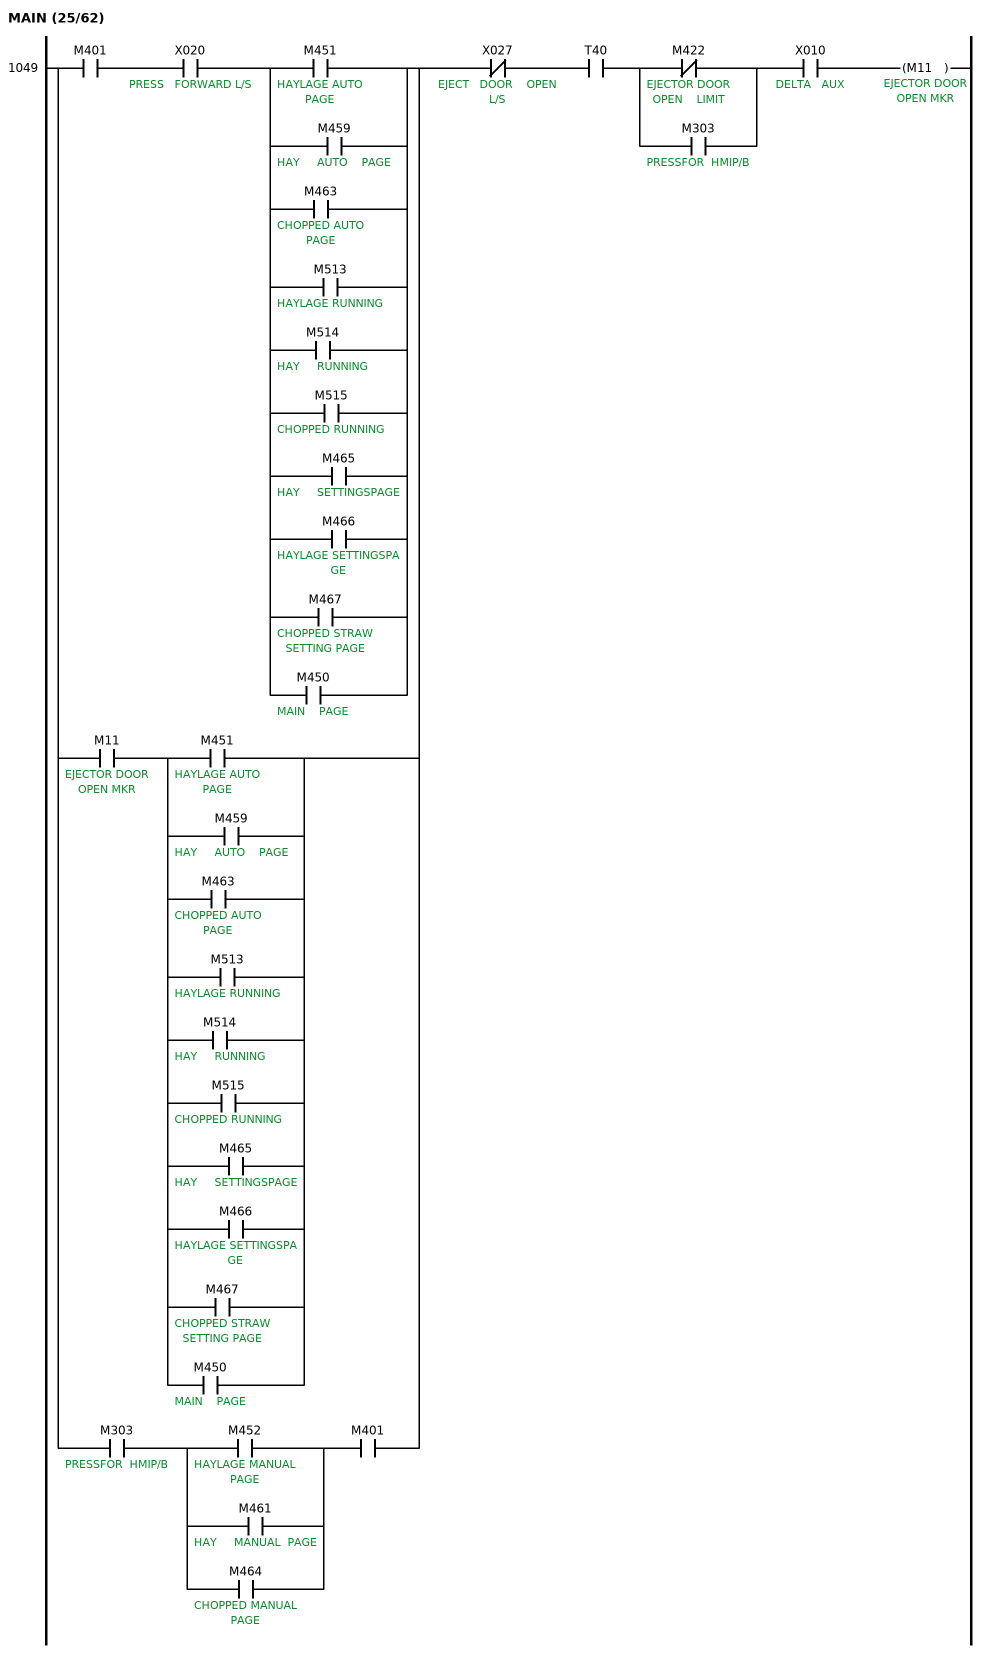
1049  LD      M401
      AND     X020  ; PRESS   FORWARD L/S
      LD      M451  ; HAYLAGE AUTO    PAGE
      OR      M459  ; HAY     AUTO    PAGE
      OR      M463  ; CHOPPED AUTO    PAGE
      OR      M513  ; HAYLAGE RUNNING
      OR      M514  ; HAY     RUNNING
      OR      M515  ; CHOPPED RUNNING
      OR      M465  ; HAY     SETTINGSPAGE
      OR      M466  ; HAYLAGE SETTINGSPAGE
      OR      M467  ; CHOPPED STRAW   SETTING PAGE
      OR      M450  ; MAIN    PAGE
      ANB
      LD      M11  ; EJECTOR DOOR    OPEN MKR
      LD      M451  ; HAYLAGE AUTO    PAGE
      OR      M459  ; HAY     AUTO    PAGE
      OR      M463  ; CHOPPED AUTO    PAGE
      OR      M513  ; HAYLAGE RUNNING
      OR      M514  ; HAY     RUNNING
      OR      M515  ; CHOPPED RUNNING
      OR      M465  ; HAY     SETTINGSPAGE
      OR      M466  ; HAYLAGE SETTINGSPAGE
      OR      M467  ; CHOPPED STRAW   SETTING PAGE
      OR      M450  ; MAIN    PAGE
      ANB
      ORB
      LD      M303  ; PRESSFOR  HMIP/B
      LD      M452  ; HAYLAGE MANUAL  PAGE
      OR      M461  ; HAY     MANUAL  PAGE
      OR      M464  ; CHOPPED MANUAL  PAGE
      ANB
      AND     M401
      ORB
      ANI     X027  ; EJECT   DOOR    OPEN L/S
      AND     T40
      LDI     M422  ; EJECTOR DOOR    OPEN    LIMIT
      OR      M303  ; PRESSFOR  HMIP/B
      ANB
      AND     X010  ; DELTA   AUX
      OUT     M11  ; EJECTOR DOOR    OPEN MKR
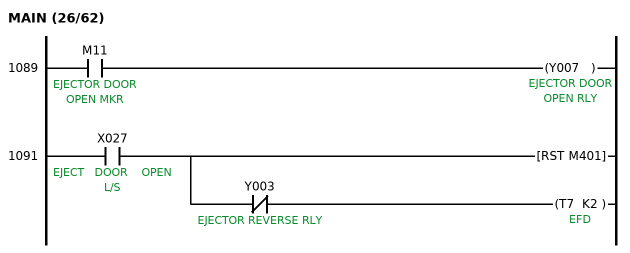
1089  LD      M11  ; EJECTOR DOOR    OPEN MKR
      OUT     Y007  ; EJECTOR DOOR    OPEN RLY
1091  LD      X027  ; EJECT   DOOR    OPEN L/S
      RST     M401
      ANI     Y003  ; EJECTOR REVERSE RLY
      OUT     T7 K2  ; EFD
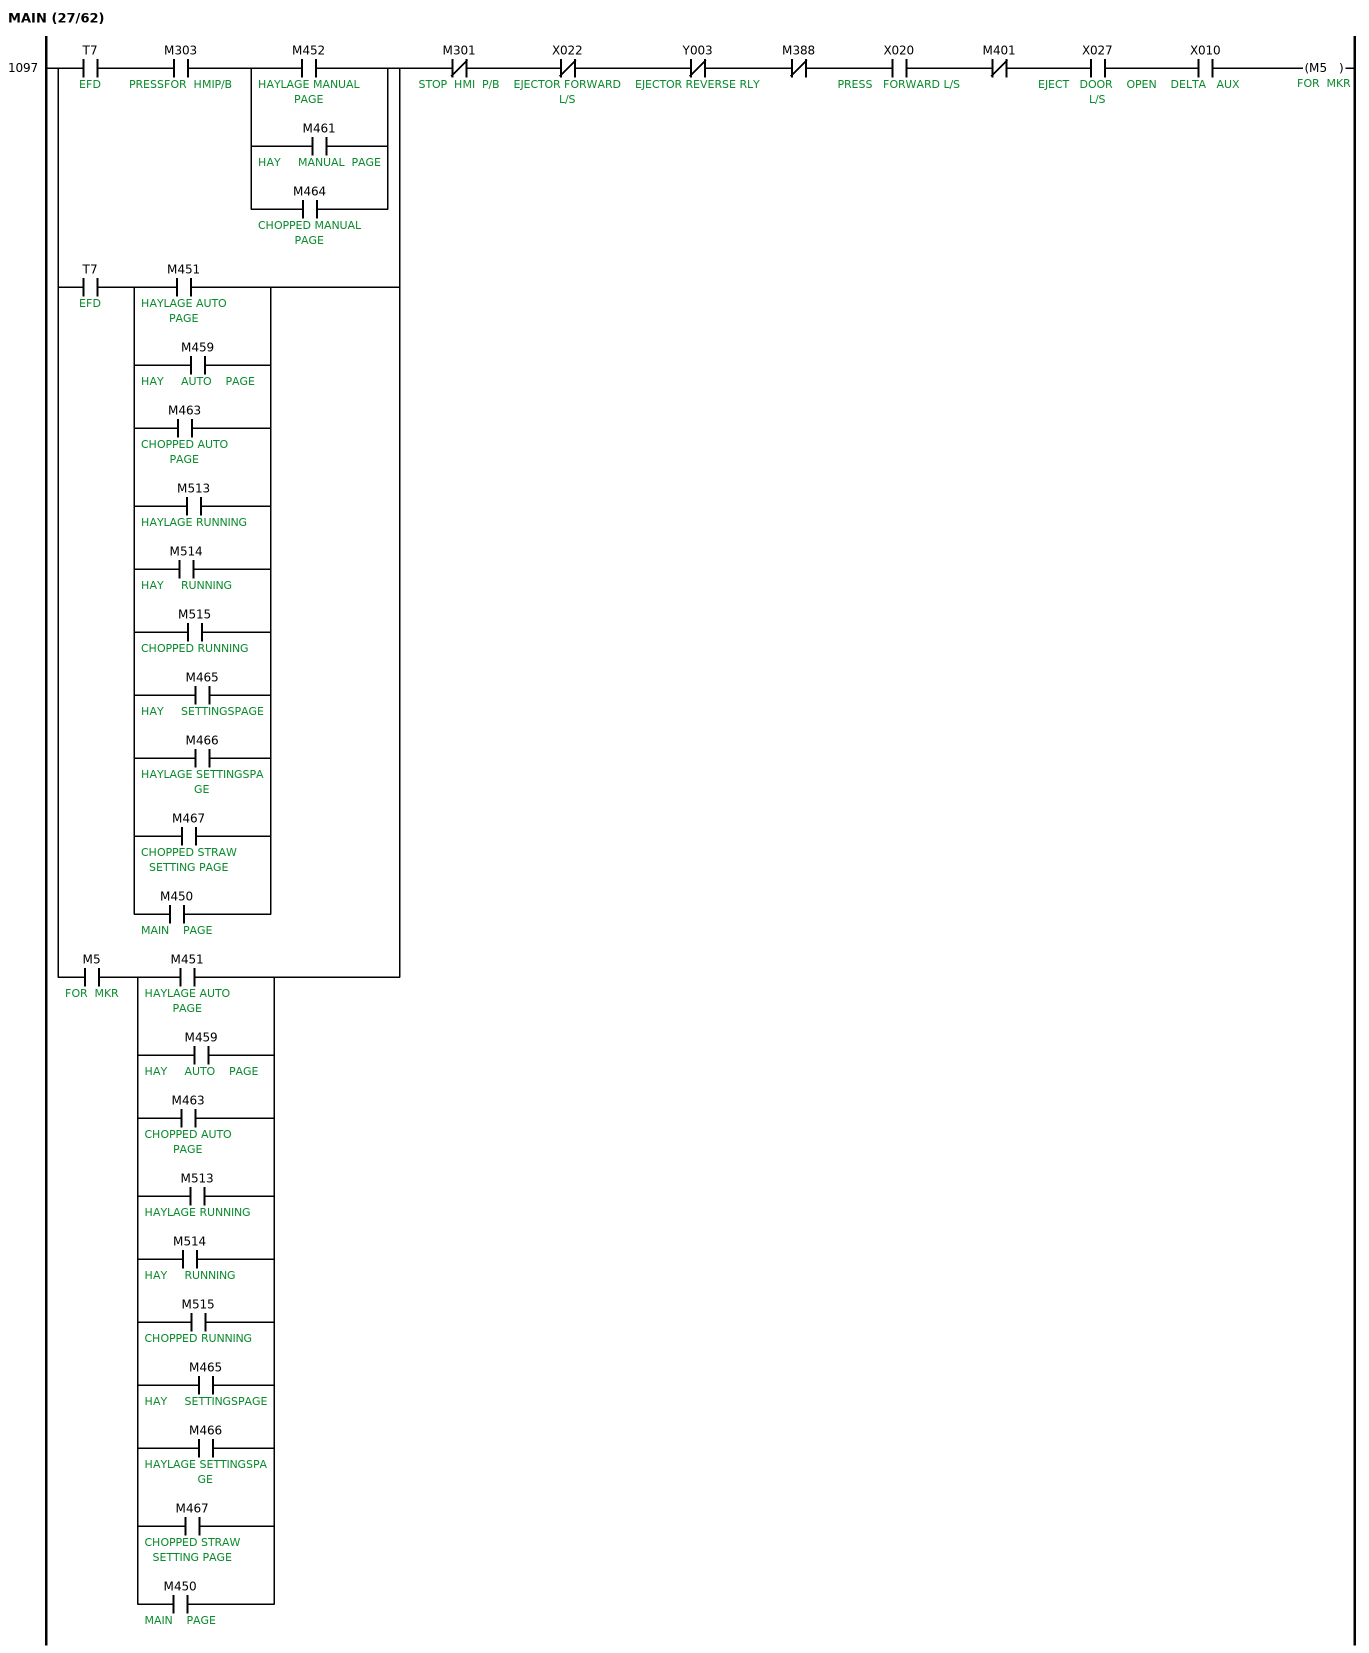
1097  LD      T7  ; EFD
      AND     M303  ; PRESSFOR  HMIP/B
      LD      M452  ; HAYLAGE MANUAL  PAGE
      OR      M461  ; HAY     MANUAL  PAGE
      OR      M464  ; CHOPPED MANUAL  PAGE
      ANB
      LD      T7  ; EFD
      LD      M451  ; HAYLAGE AUTO    PAGE
      OR      M459  ; HAY     AUTO    PAGE
      OR      M463  ; CHOPPED AUTO    PAGE
      OR      M513  ; HAYLAGE RUNNING
      OR      M514  ; HAY     RUNNING
      OR      M515  ; CHOPPED RUNNING
      OR      M465  ; HAY     SETTINGSPAGE
      OR      M466  ; HAYLAGE SETTINGSPAGE
      OR      M467  ; CHOPPED STRAW   SETTING PAGE
      OR      M450  ; MAIN    PAGE
      ANB
      ORB
      LD      M5  ; FOR  MKR
      LD      M451  ; HAYLAGE AUTO    PAGE
      OR      M459  ; HAY     AUTO    PAGE
      OR      M463  ; CHOPPED AUTO    PAGE
      OR      M513  ; HAYLAGE RUNNING
      OR      M514  ; HAY     RUNNING
      OR      M515  ; CHOPPED RUNNING
      OR      M465  ; HAY     SETTINGSPAGE
      OR      M466  ; HAYLAGE SETTINGSPAGE
      OR      M467  ; CHOPPED STRAW   SETTING PAGE
      OR      M450  ; MAIN    PAGE
      ANB
      ORB
      ANI     M301  ; STOP  HMI  P/B
      ANI     X022  ; EJECTOR FORWARD L/S
      ANI     Y003  ; EJECTOR REVERSE RLY
      ANI     M388
      AND     X020  ; PRESS   FORWARD L/S
      ANI     M401
      AND     X027  ; EJECT   DOOR    OPEN L/S
      AND     X010  ; DELTA   AUX
      OUT     M5  ; FOR  MKR
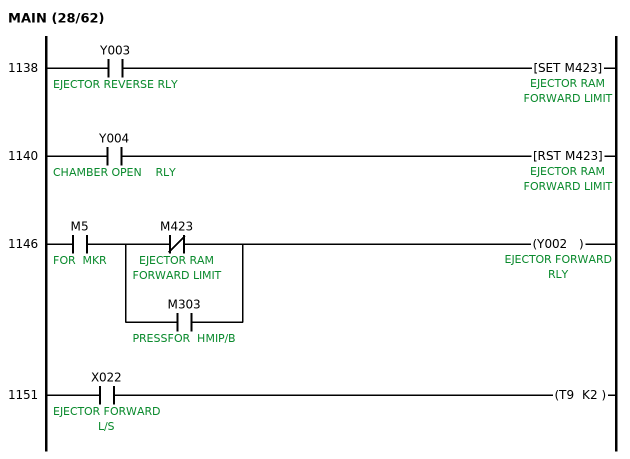
1138  LD      Y003  ; EJECTOR REVERSE RLY
      SET     M423  ; EJECTOR RAM     FORWARD LIMIT
1140  LD      Y004  ; CHAMBER OPEN    RLY
      RST     M423  ; EJECTOR RAM     FORWARD LIMIT
1146  LD      M5  ; FOR  MKR
      LDI     M423  ; EJECTOR RAM     FORWARD LIMIT
      OR      M303  ; PRESSFOR  HMIP/B
      ANB
      OUT     Y002  ; EJECTOR FORWARD RLY
1151  LD      X022  ; EJECTOR FORWARD L/S
      OUT     T9 K2
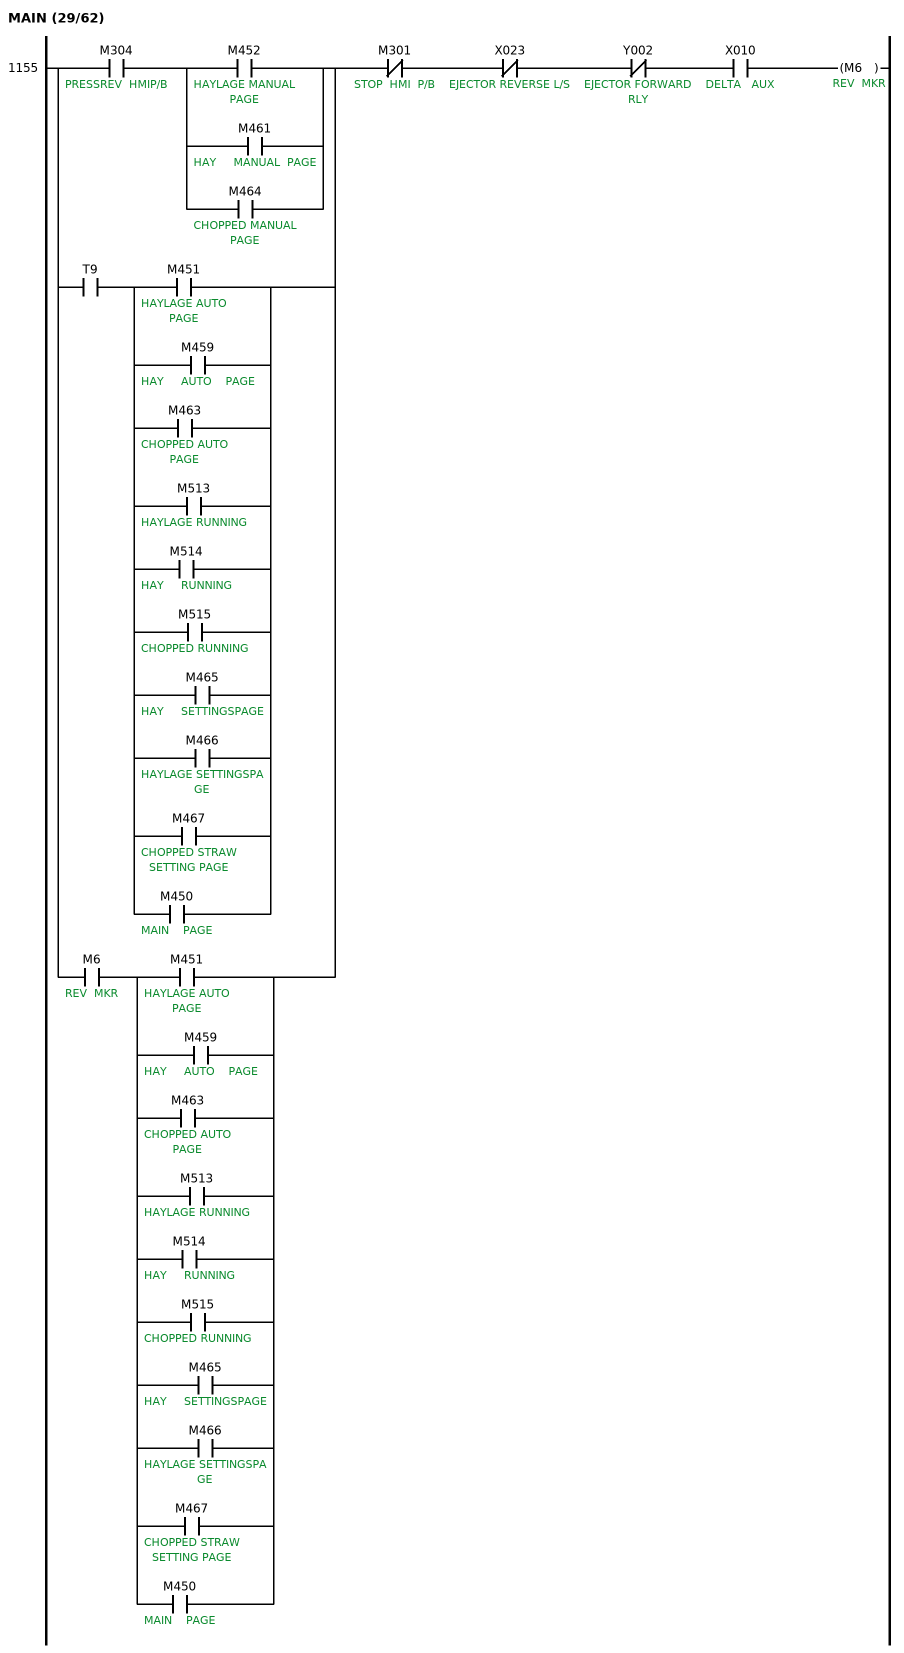
1155  LD      M304  ; PRESSREV  HMIP/B
      LD      M452  ; HAYLAGE MANUAL  PAGE
      OR      M461  ; HAY     MANUAL  PAGE
      OR      M464  ; CHOPPED MANUAL  PAGE
      ANB
      LD      T9
      LD      M451  ; HAYLAGE AUTO    PAGE
      OR      M459  ; HAY     AUTO    PAGE
      OR      M463  ; CHOPPED AUTO    PAGE
      OR      M513  ; HAYLAGE RUNNING
      OR      M514  ; HAY     RUNNING
      OR      M515  ; CHOPPED RUNNING
      OR      M465  ; HAY     SETTINGSPAGE
      OR      M466  ; HAYLAGE SETTINGSPAGE
      OR      M467  ; CHOPPED STRAW   SETTING PAGE
      OR      M450  ; MAIN    PAGE
      ANB
      ORB
      LD      M6  ; REV  MKR
      LD      M451  ; HAYLAGE AUTO    PAGE
      OR      M459  ; HAY     AUTO    PAGE
      OR      M463  ; CHOPPED AUTO    PAGE
      OR      M513  ; HAYLAGE RUNNING
      OR      M514  ; HAY     RUNNING
      OR      M515  ; CHOPPED RUNNING
      OR      M465  ; HAY     SETTINGSPAGE
      OR      M466  ; HAYLAGE SETTINGSPAGE
      OR      M467  ; CHOPPED STRAW   SETTING PAGE
      OR      M450  ; MAIN    PAGE
      ANB
      ORB
      ANI     M301  ; STOP  HMI  P/B
      ANI     X023  ; EJECTOR REVERSE L/S
      ANI     Y002  ; EJECTOR FORWARD RLY
      AND     X010  ; DELTA   AUX
      OUT     M6  ; REV  MKR
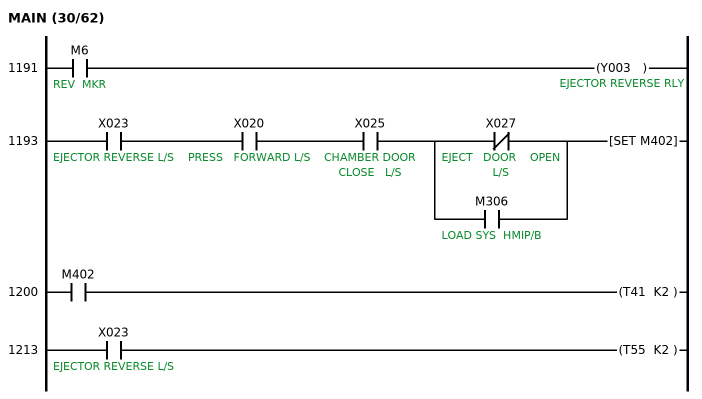
1191  LD      M6  ; REV  MKR
      OUT     Y003  ; EJECTOR REVERSE RLY
1193  LD      X023  ; EJECTOR REVERSE L/S
      AND     X020  ; PRESS   FORWARD L/S
      AND     X025  ; CHAMBER DOOR    CLOSE   L/S
      LDI     X027  ; EJECT   DOOR    OPEN L/S
      OR      M306  ; LOAD SYS  HMIP/B
      ANB
      SET     M402
1200  LD      M402
      OUT     T41 K2
1213  LD      X023  ; EJECTOR REVERSE L/S
      OUT     T55 K2
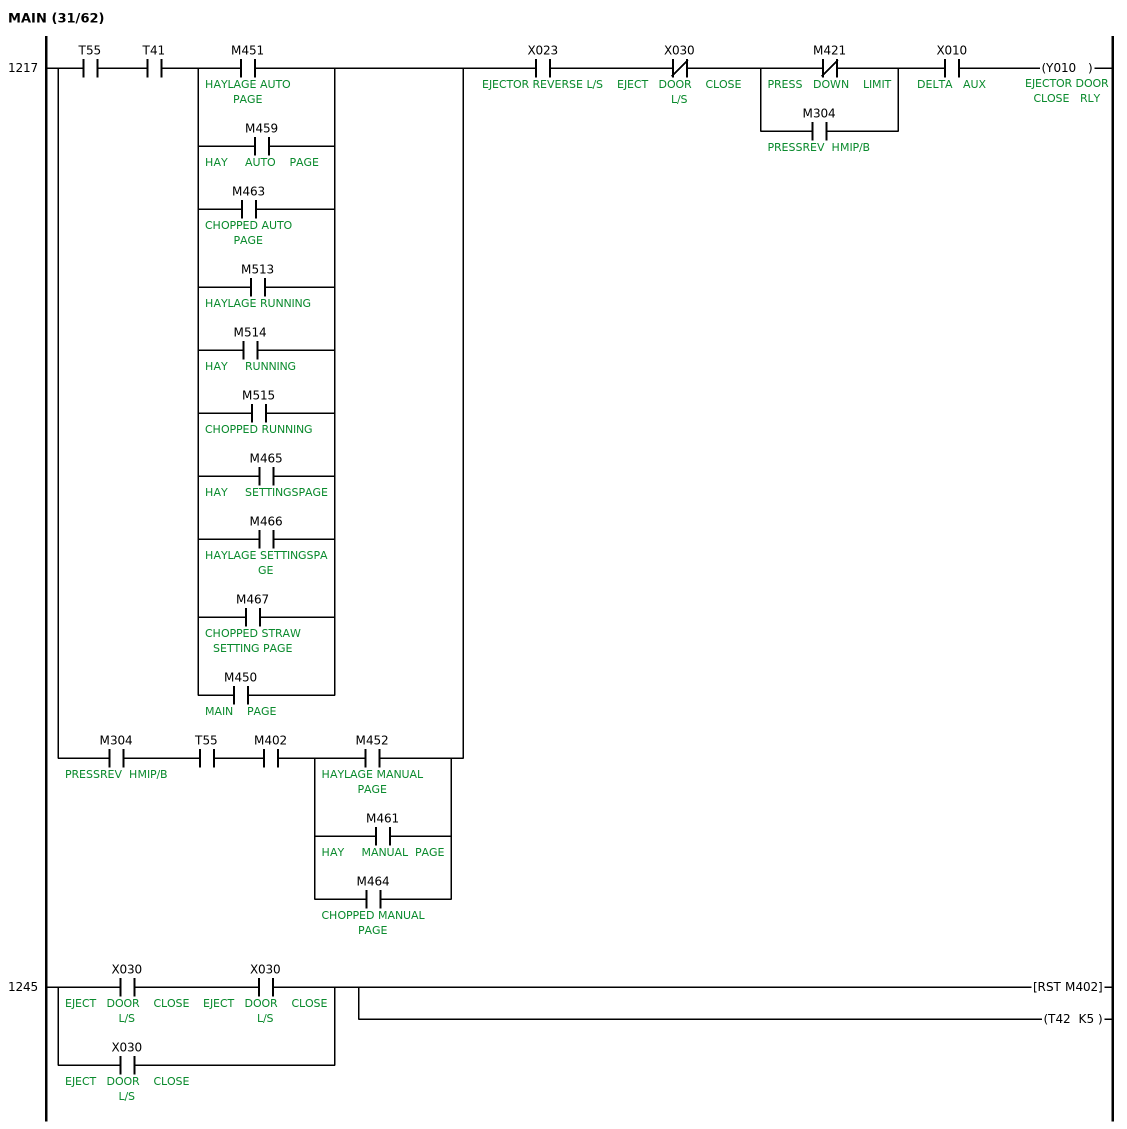
1217  LD      T55
      AND     T41
      LD      M451  ; HAYLAGE AUTO    PAGE
      OR      M459  ; HAY     AUTO    PAGE
      OR      M463  ; CHOPPED AUTO    PAGE
      OR      M513  ; HAYLAGE RUNNING
      OR      M514  ; HAY     RUNNING
      OR      M515  ; CHOPPED RUNNING
      OR      M465  ; HAY     SETTINGSPAGE
      OR      M466  ; HAYLAGE SETTINGSPAGE
      OR      M467  ; CHOPPED STRAW   SETTING PAGE
      OR      M450  ; MAIN    PAGE
      ANB
      LD      M304  ; PRESSREV  HMIP/B
      AND     T55
      AND     M402
      LD      M452  ; HAYLAGE MANUAL  PAGE
      OR      M461  ; HAY     MANUAL  PAGE
      OR      M464  ; CHOPPED MANUAL  PAGE
      ANB
      ORB
      AND     X023  ; EJECTOR REVERSE L/S
      ANI     X030  ; EJECT   DOOR    CLOSE L/S
      LDI     M421  ; PRESS   DOWN    LIMIT
      OR      M304  ; PRESSREV  HMIP/B
      ANB
      AND     X010  ; DELTA   AUX
      OUT     Y010  ; EJECTOR DOOR    CLOSE   RLY
1245  LD      X030  ; EJECT   DOOR    CLOSE L/S
      AND     X030  ; EJECT   DOOR    CLOSE L/S
      OR      X030  ; EJECT   DOOR    CLOSE L/S
      RST     M402
      OUT     T42 K5
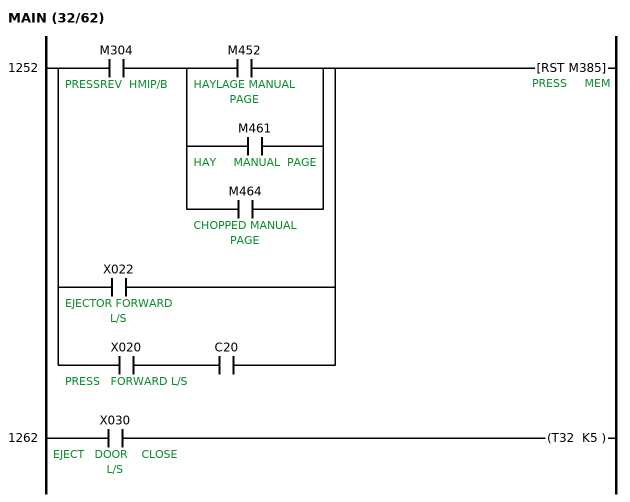
1252  LD      M304  ; PRESSREV  HMIP/B
      LD      M452  ; HAYLAGE MANUAL  PAGE
      OR      M461  ; HAY     MANUAL  PAGE
      OR      M464  ; CHOPPED MANUAL  PAGE
      ANB
      OR      X022  ; EJECTOR FORWARD L/S
      LD      X020  ; PRESS   FORWARD L/S
      AND     C20
      ORB
      RST     M385  ; PRESS     MEM
1262  LD      X030  ; EJECT   DOOR    CLOSE L/S
      OUT     T32 K5
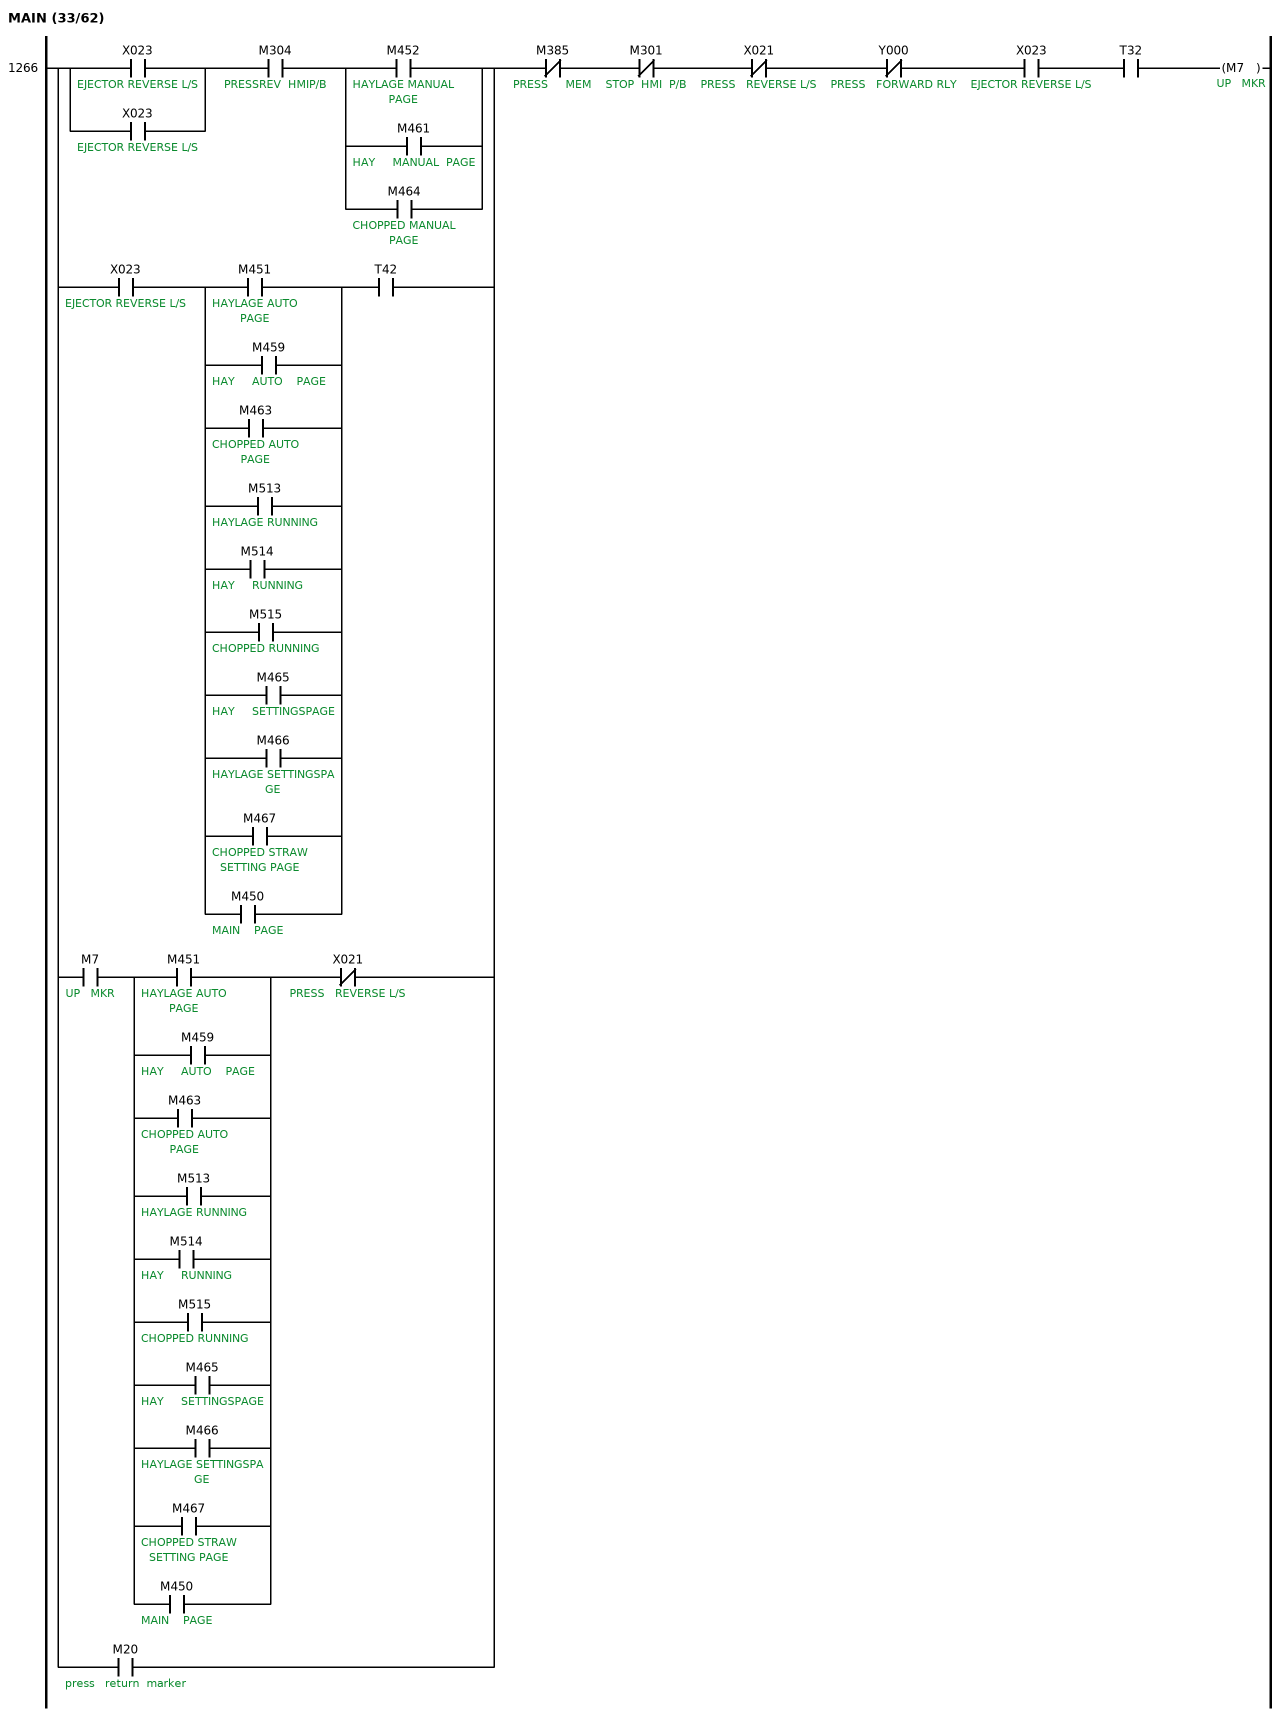
1266  LD      X023  ; EJECTOR REVERSE L/S
      OR      X023  ; EJECTOR REVERSE L/S
      AND     M304  ; PRESSREV  HMIP/B
      LD      M452  ; HAYLAGE MANUAL  PAGE
      OR      M461  ; HAY     MANUAL  PAGE
      OR      M464  ; CHOPPED MANUAL  PAGE
      ANB
      LD      X023  ; EJECTOR REVERSE L/S
      LD      M451  ; HAYLAGE AUTO    PAGE
      OR      M459  ; HAY     AUTO    PAGE
      OR      M463  ; CHOPPED AUTO    PAGE
      OR      M513  ; HAYLAGE RUNNING
      OR      M514  ; HAY     RUNNING
      OR      M515  ; CHOPPED RUNNING
      OR      M465  ; HAY     SETTINGSPAGE
      OR      M466  ; HAYLAGE SETTINGSPAGE
      OR      M467  ; CHOPPED STRAW   SETTING PAGE
      OR      M450  ; MAIN    PAGE
      ANB
      AND     T42
      ORB
      LD      M7  ; UP   MKR
      LD      M451  ; HAYLAGE AUTO    PAGE
      OR      M459  ; HAY     AUTO    PAGE
      OR      M463  ; CHOPPED AUTO    PAGE
      OR      M513  ; HAYLAGE RUNNING
      OR      M514  ; HAY     RUNNING
      OR      M515  ; CHOPPED RUNNING
      OR      M465  ; HAY     SETTINGSPAGE
      OR      M466  ; HAYLAGE SETTINGSPAGE
      OR      M467  ; CHOPPED STRAW   SETTING PAGE
      OR      M450  ; MAIN    PAGE
      ANB
      ANI     X021  ; PRESS   REVERSE L/S
      ORB
      OR      M20  ; press   return  marker
      ANI     M385  ; PRESS     MEM
      ANI     M301  ; STOP  HMI  P/B
      ANI     X021  ; PRESS   REVERSE L/S
      ANI     Y000  ; PRESS   FORWARD RLY
      AND     X023  ; EJECTOR REVERSE L/S
      AND     T32
      OUT     M7  ; UP   MKR
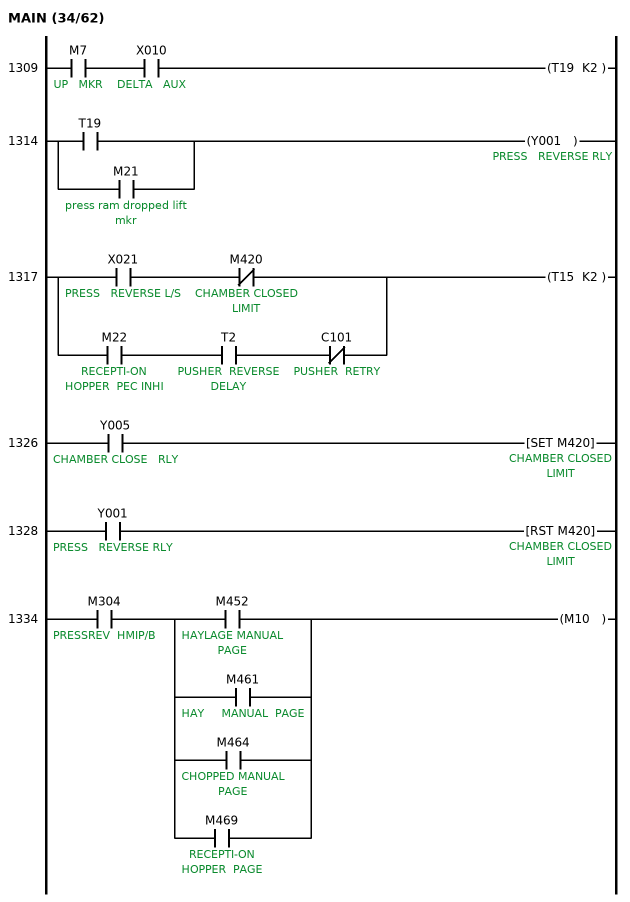
1309  LD      M7  ; UP   MKR
      AND     X010  ; DELTA   AUX
      OUT     T19 K2
1314  LD      T19
      OR      M21  ; press ram dropped lift mkr
      OUT     Y001  ; PRESS   REVERSE RLY
1317  LD      X021  ; PRESS   REVERSE L/S
      ANI     M420  ; CHAMBER CLOSED  LIMIT
      LD      M22  ; RECEPTI-ON      HOPPER  PEC INHI
      AND     T2  ; PUSHER  REVERSE DELAY
      ANI     C101  ; PUSHER  RETRY
      ORB
      OUT     T15 K2
1326  LD      Y005  ; CHAMBER CLOSE   RLY
      SET     M420  ; CHAMBER CLOSED  LIMIT
1328  LD      Y001  ; PRESS   REVERSE RLY
      RST     M420  ; CHAMBER CLOSED  LIMIT
1334  LD      M304  ; PRESSREV  HMIP/B
      LD      M452  ; HAYLAGE MANUAL  PAGE
      OR      M461  ; HAY     MANUAL  PAGE
      OR      M464  ; CHOPPED MANUAL  PAGE
      OR      M469  ; RECEPTI-ON      HOPPER  PAGE
      ANB
      OUT     M10
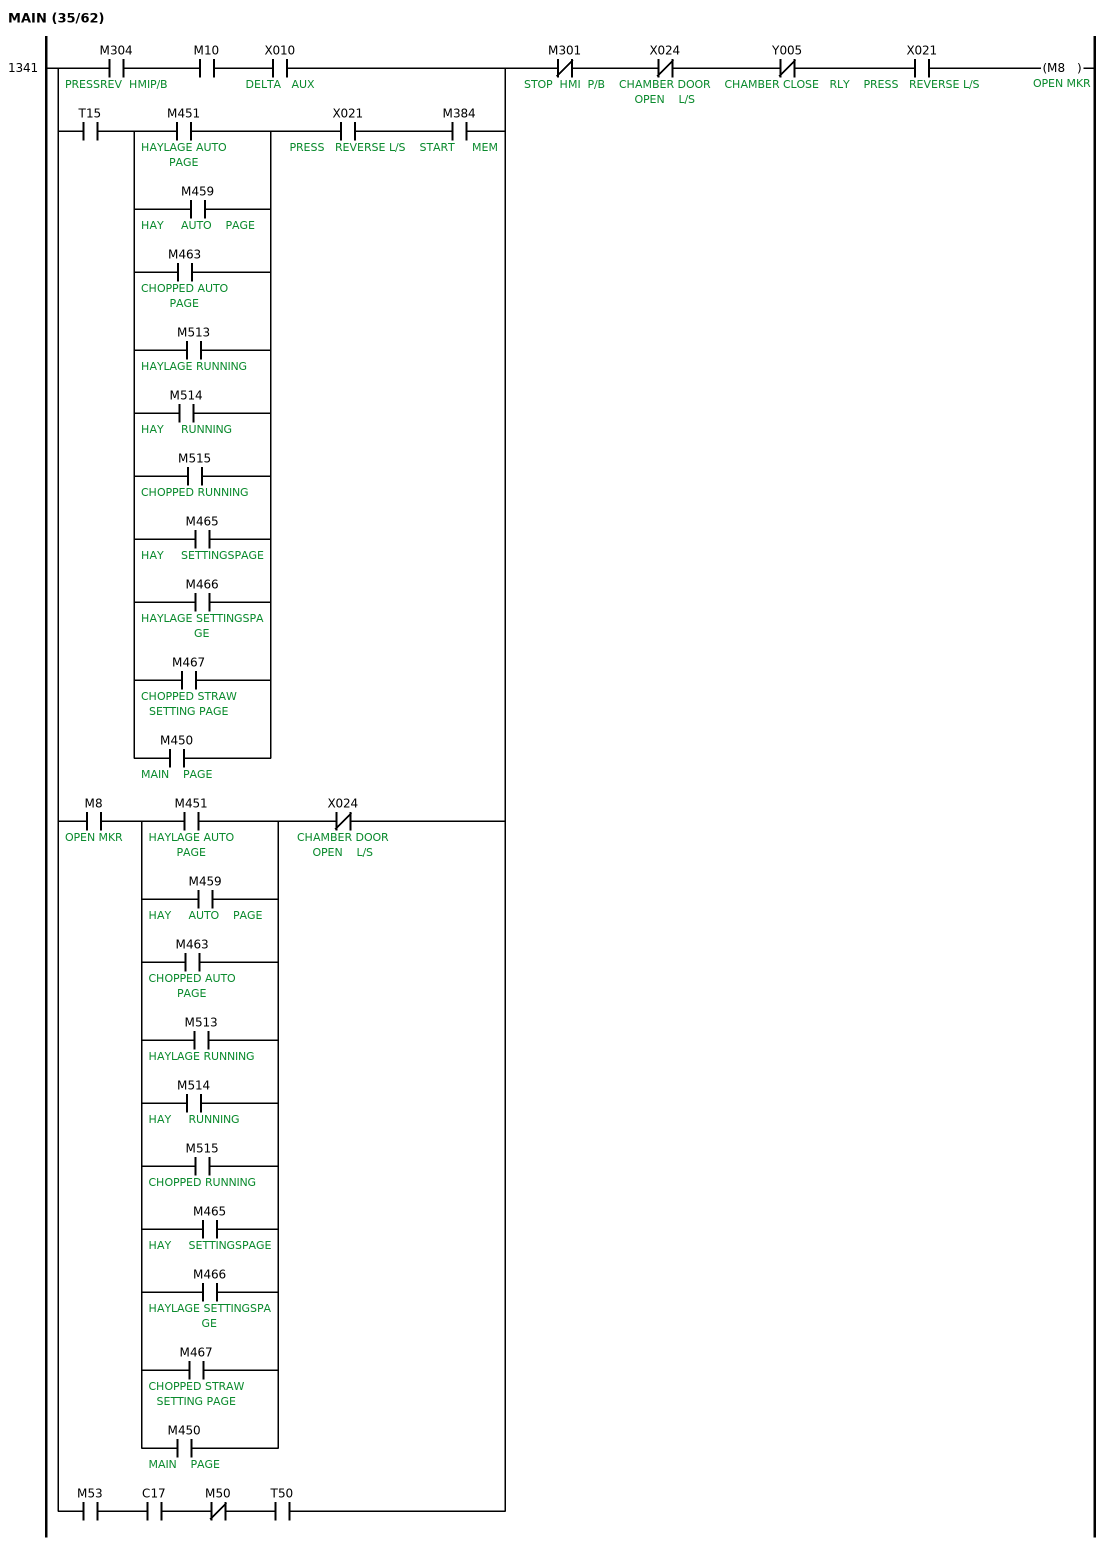
1341  LD      M304  ; PRESSREV  HMIP/B
      AND     M10
      AND     X010  ; DELTA   AUX
      LD      T15
      LD      M451  ; HAYLAGE AUTO    PAGE
      OR      M459  ; HAY     AUTO    PAGE
      OR      M463  ; CHOPPED AUTO    PAGE
      OR      M513  ; HAYLAGE RUNNING
      OR      M514  ; HAY     RUNNING
      OR      M515  ; CHOPPED RUNNING
      OR      M465  ; HAY     SETTINGSPAGE
      OR      M466  ; HAYLAGE SETTINGSPAGE
      OR      M467  ; CHOPPED STRAW   SETTING PAGE
      OR      M450  ; MAIN    PAGE
      ANB
      AND     X021  ; PRESS   REVERSE L/S
      AND     M384  ; START     MEM
      ORB
      LD      M8  ; OPEN MKR
      LD      M451  ; HAYLAGE AUTO    PAGE
      OR      M459  ; HAY     AUTO    PAGE
      OR      M463  ; CHOPPED AUTO    PAGE
      OR      M513  ; HAYLAGE RUNNING
      OR      M514  ; HAY     RUNNING
      OR      M515  ; CHOPPED RUNNING
      OR      M465  ; HAY     SETTINGSPAGE
      OR      M466  ; HAYLAGE SETTINGSPAGE
      OR      M467  ; CHOPPED STRAW   SETTING PAGE
      OR      M450  ; MAIN    PAGE
      ANB
      ANI     X024  ; CHAMBER DOOR    OPEN    L/S
      ORB
      LD      M53
      AND     C17
      ANI     M50
      AND     T50
      ORB
      ANI     M301  ; STOP  HMI  P/B
      ANI     X024  ; CHAMBER DOOR    OPEN    L/S
      ANI     Y005  ; CHAMBER CLOSE   RLY
      AND     X021  ; PRESS   REVERSE L/S
      OUT     M8  ; OPEN MKR
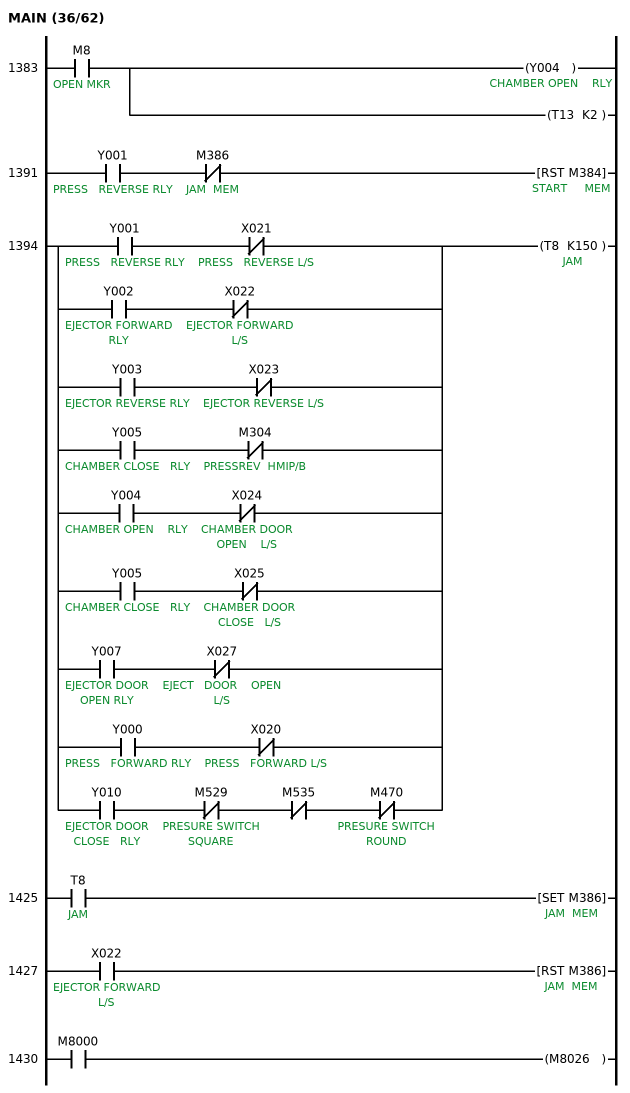
1383  LD      M8  ; OPEN MKR
      OUT     Y004  ; CHAMBER OPEN    RLY
      OUT     T13 K2
1391  LD      Y001  ; PRESS   REVERSE RLY
      ANI     M386  ; JAM  MEM
      RST     M384  ; START     MEM
1394  LD      Y001  ; PRESS   REVERSE RLY
      ANI     X021  ; PRESS   REVERSE L/S
      LD      Y002  ; EJECTOR FORWARD RLY
      ANI     X022  ; EJECTOR FORWARD L/S
      ORB
      LD      Y003  ; EJECTOR REVERSE RLY
      ANI     X023  ; EJECTOR REVERSE L/S
      ORB
      LD      Y005  ; CHAMBER CLOSE   RLY
      ANI     M304  ; PRESSREV  HMIP/B
      ORB
      LD      Y004  ; CHAMBER OPEN    RLY
      ANI     X024  ; CHAMBER DOOR    OPEN    L/S
      ORB
      LD      Y005  ; CHAMBER CLOSE   RLY
      ANI     X025  ; CHAMBER DOOR    CLOSE   L/S
      ORB
      LD      Y007  ; EJECTOR DOOR    OPEN RLY
      ANI     X027  ; EJECT   DOOR    OPEN L/S
      ORB
      LD      Y000  ; PRESS   FORWARD RLY
      ANI     X020  ; PRESS   FORWARD L/S
      ORB
      LD      Y010  ; EJECTOR DOOR    CLOSE   RLY
      ANI     M529  ; PRESURE SWITCH  SQUARE
      ANI     M535
      ANI     M470  ; PRESURE SWITCH  ROUND
      ORB
      OUT     T8 K150  ; JAM
1425  LD      T8  ; JAM
      SET     M386  ; JAM  MEM
1427  LD      X022  ; EJECTOR FORWARD L/S
      RST     M386  ; JAM  MEM
1430  LD      M8000
      OUT     M8026
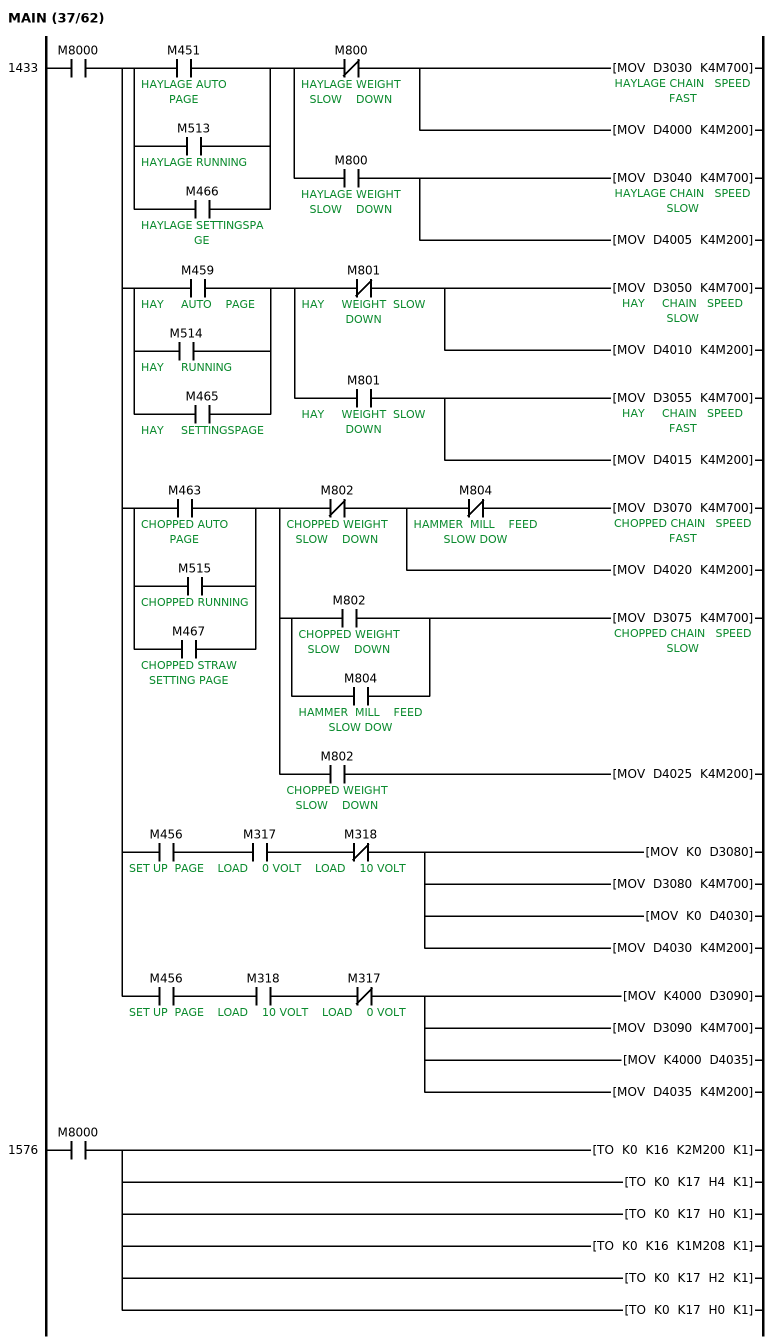
1433  LD      M8000
      MPS
      LD      M451  ; HAYLAGE AUTO    PAGE
      OR      M513  ; HAYLAGE RUNNING
      OR      M466  ; HAYLAGE SETTINGSPAGE
      ANB
      MPS
      ANI     M800  ; HAYLAGE WEIGHT  SLOW    DOWN
      MOV     D3030 K4M700  ; HAYLAGE CHAIN   SPEED   FAST
      MOV     D4000 K4M200
      MPP
      AND     M800  ; HAYLAGE WEIGHT  SLOW    DOWN
      MOV     D3040 K4M700  ; HAYLAGE CHAIN   SPEED   SLOW
      MOV     D4005 K4M200
      MRD
      LD      M459  ; HAY     AUTO    PAGE
      OR      M514  ; HAY     RUNNING
      OR      M465  ; HAY     SETTINGSPAGE
      ANB
      MPS
      ANI     M801  ; HAY     WEIGHT  SLOW    DOWN
      MOV     D3050 K4M700  ; HAY     CHAIN   SPEED   SLOW
      MOV     D4010 K4M200
      MPP
      AND     M801  ; HAY     WEIGHT  SLOW    DOWN
      MOV     D3055 K4M700  ; HAY     CHAIN   SPEED   FAST
      MOV     D4015 K4M200
      MRD
      LD      M463  ; CHOPPED AUTO    PAGE
      OR      M515  ; CHOPPED RUNNING
      OR      M467  ; CHOPPED STRAW   SETTING PAGE
      ANB
      MPS
      ANI     M802  ; CHOPPED WEIGHT  SLOW    DOWN
      MPS
      ANI     M804  ; HAMMER  MILL    FEED    SLOW DOW
      MOV     D3070 K4M700  ; CHOPPED CHAIN   SPEED   FAST
      MPP
      MOV     D4020 K4M200
      MRD
      LD      M802  ; CHOPPED WEIGHT  SLOW    DOWN
      OR      M804  ; HAMMER  MILL    FEED    SLOW DOW
      ANB
      MOV     D3075 K4M700  ; CHOPPED CHAIN   SPEED   SLOW
      MPP
      AND     M802  ; CHOPPED WEIGHT  SLOW    DOWN
      MOV     D4025 K4M200
      MRD
      AND     M456  ; SET UP  PAGE
      AND     M317  ; LOAD    0 VOLT
      ANI     M318  ; LOAD    10 VOLT
      MOV     K0 D3080
      MOV     D3080 K4M700
      MOV     K0 D4030
      MOV     D4030 K4M200
      MPP
      AND     M456  ; SET UP  PAGE
      AND     M318  ; LOAD    10 VOLT
      ANI     M317  ; LOAD    0 VOLT
      MOV     K4000 D3090
      MOV     D3090 K4M700
      MOV     K4000 D4035
      MOV     D4035 K4M200
1576  LD      M8000
      TO      K0 K16 K2M200 K1
      TO      K0 K17 H4 K1
      TO      K0 K17 H0 K1
      TO      K0 K16 K1M208 K1
      TO      K0 K17 H2 K1
      TO      K0 K17 H0 K1
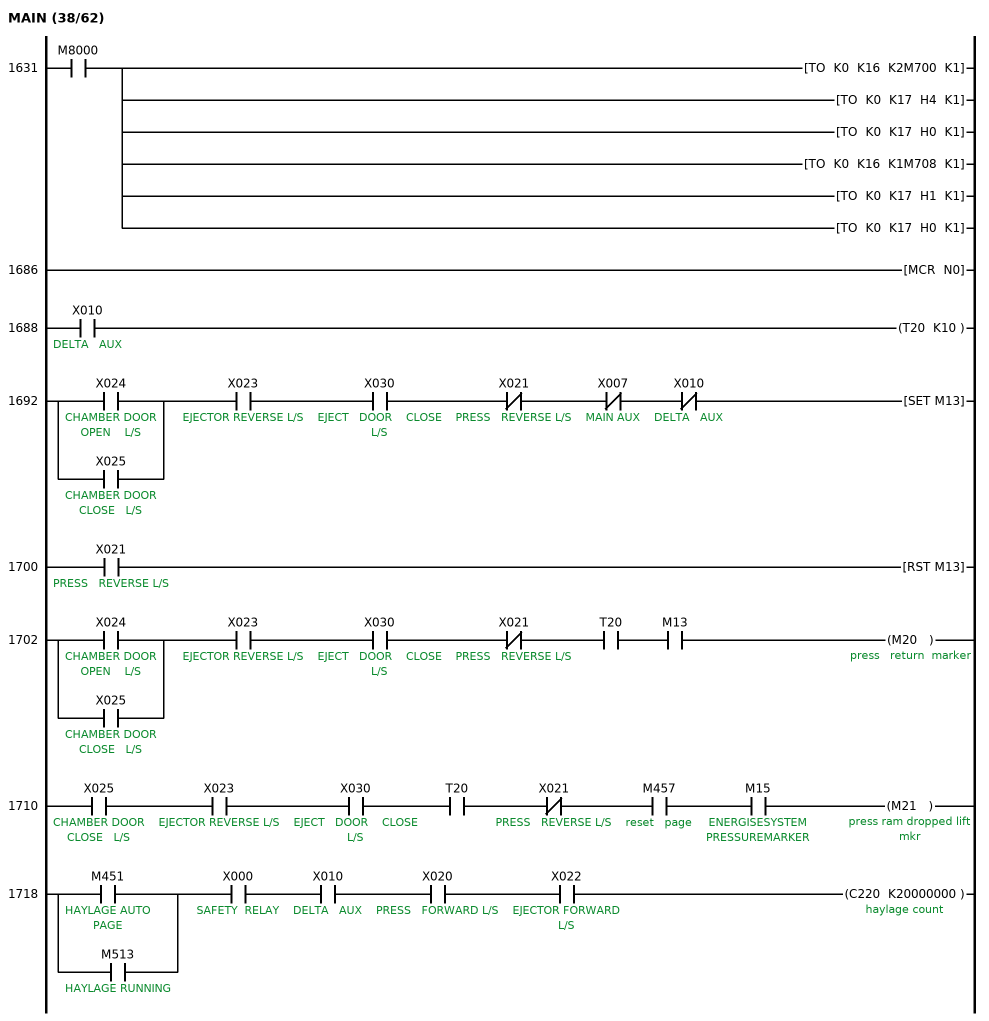
1631  LD      M8000
      TO      K0 K16 K2M700 K1
      TO      K0 K17 H4 K1
      TO      K0 K17 H0 K1
      TO      K0 K16 K1M708 K1
      TO      K0 K17 H1 K1
      TO      K0 K17 H0 K1
1686  MCR     N0
1688  LD      X010  ; DELTA   AUX
      OUT     T20 K10
1692  LD      X024  ; CHAMBER DOOR    OPEN    L/S
      OR      X025  ; CHAMBER DOOR    CLOSE   L/S
      AND     X023  ; EJECTOR REVERSE L/S
      AND     X030  ; EJECT   DOOR    CLOSE L/S
      ANI     X021  ; PRESS   REVERSE L/S
      ANI     X007  ; MAIN AUX
      ANI     X010  ; DELTA   AUX
      SET     M13
1700  LD      X021  ; PRESS   REVERSE L/S
      RST     M13
1702  LD      X024  ; CHAMBER DOOR    OPEN    L/S
      OR      X025  ; CHAMBER DOOR    CLOSE   L/S
      AND     X023  ; EJECTOR REVERSE L/S
      AND     X030  ; EJECT   DOOR    CLOSE L/S
      ANI     X021  ; PRESS   REVERSE L/S
      AND     T20
      AND     M13
      OUT     M20  ; press   return  marker
1710  LD      X025  ; CHAMBER DOOR    CLOSE   L/S
      AND     X023  ; EJECTOR REVERSE L/S
      AND     X030  ; EJECT   DOOR    CLOSE L/S
      AND     T20
      ANI     X021  ; PRESS   REVERSE L/S
      AND     M457  ; reset   page
      AND     M15  ; ENERGISESYSTEM  PRESSUREMARKER
      OUT     M21  ; press ram dropped lift mkr
1718  LD      M451  ; HAYLAGE AUTO    PAGE
      OR      M513  ; HAYLAGE RUNNING
      AND     X000  ; SAFETY  RELAY
      AND     X010  ; DELTA   AUX
      AND     X020  ; PRESS   FORWARD L/S
      AND     X022  ; EJECTOR FORWARD L/S
      OUT     C220 K20000000  ; haylage count
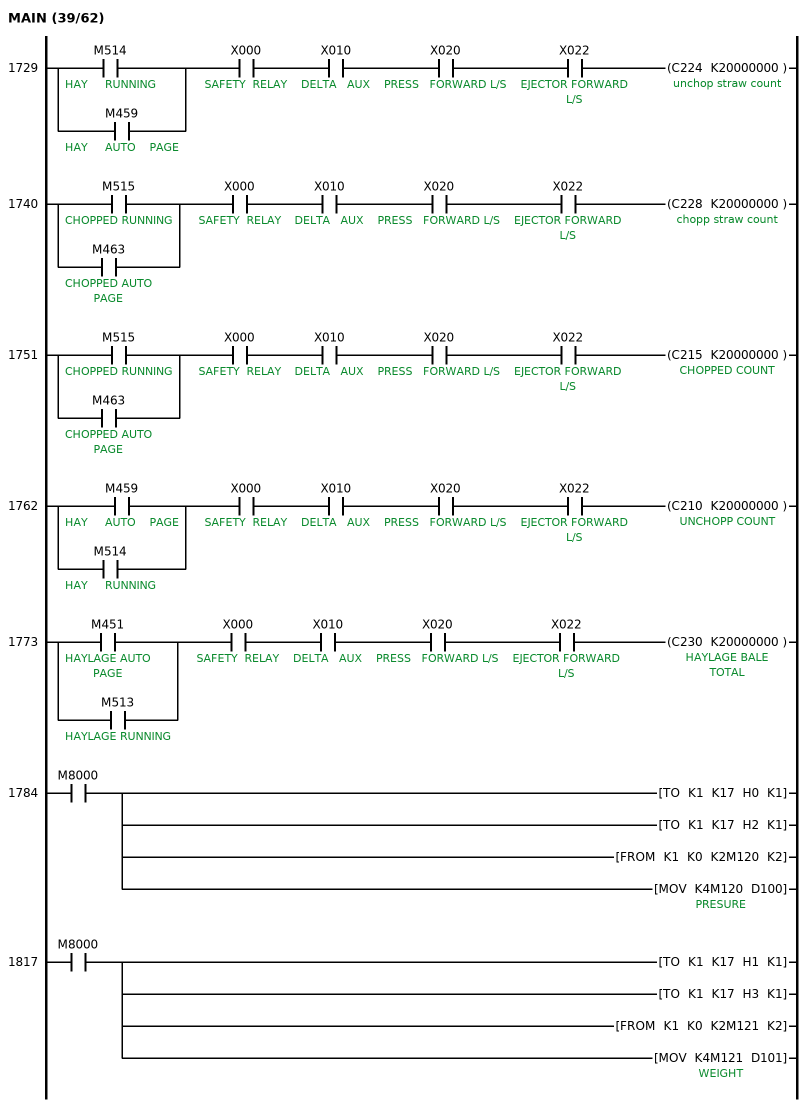
1729  LD      M514  ; HAY     RUNNING
      OR      M459  ; HAY     AUTO    PAGE
      AND     X000  ; SAFETY  RELAY
      AND     X010  ; DELTA   AUX
      AND     X020  ; PRESS   FORWARD L/S
      AND     X022  ; EJECTOR FORWARD L/S
      OUT     C224 K20000000  ; unchop straw count
1740  LD      M515  ; CHOPPED RUNNING
      OR      M463  ; CHOPPED AUTO    PAGE
      AND     X000  ; SAFETY  RELAY
      AND     X010  ; DELTA   AUX
      AND     X020  ; PRESS   FORWARD L/S
      AND     X022  ; EJECTOR FORWARD L/S
      OUT     C228 K20000000  ; chopp straw count
1751  LD      M515  ; CHOPPED RUNNING
      OR      M463  ; CHOPPED AUTO    PAGE
      AND     X000  ; SAFETY  RELAY
      AND     X010  ; DELTA   AUX
      AND     X020  ; PRESS   FORWARD L/S
      AND     X022  ; EJECTOR FORWARD L/S
      OUT     C215 K20000000  ; CHOPPED COUNT
1762  LD      M459  ; HAY     AUTO    PAGE
      OR      M514  ; HAY     RUNNING
      AND     X000  ; SAFETY  RELAY
      AND     X010  ; DELTA   AUX
      AND     X020  ; PRESS   FORWARD L/S
      AND     X022  ; EJECTOR FORWARD L/S
      OUT     C210 K20000000  ; UNCHOPP COUNT
1773  LD      M451  ; HAYLAGE AUTO    PAGE
      OR      M513  ; HAYLAGE RUNNING
      AND     X000  ; SAFETY  RELAY
      AND     X010  ; DELTA   AUX
      AND     X020  ; PRESS   FORWARD L/S
      AND     X022  ; EJECTOR FORWARD L/S
      OUT     C230 K20000000  ; HAYLAGE BALE    TOTAL
1784  LD      M8000
      TO      K1 K17 H0 K1
      TO      K1 K17 H2 K1
      FROM    K1 K0 K2M120 K2
      MOV     K4M120 D100  ; PRESURE
1817  LD      M8000
      TO      K1 K17 H1 K1
      TO      K1 K17 H3 K1
      FROM    K1 K0 K2M121 K2
      MOV     K4M121 D101  ; WEIGHT
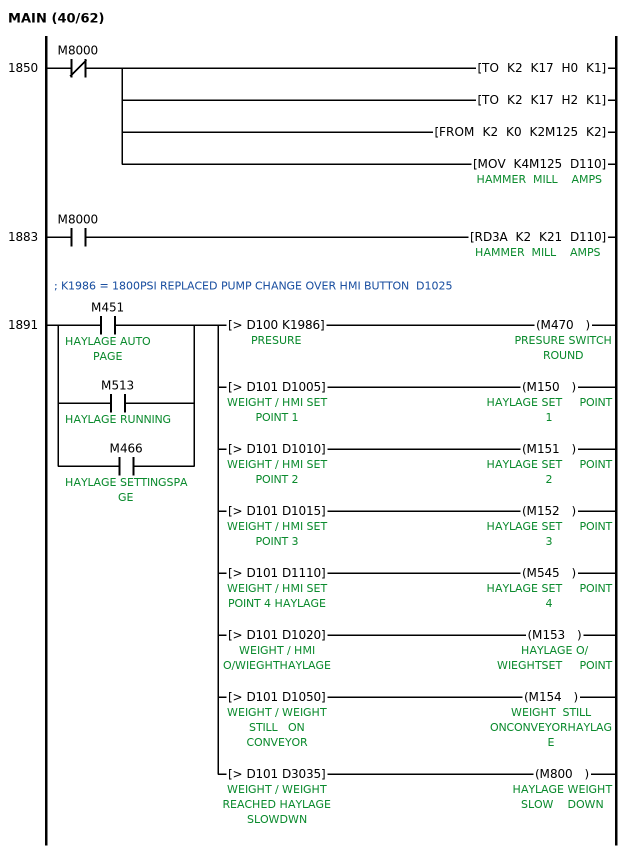
1850  LDI     M8000
      TO      K2 K17 H0 K1
      TO      K2 K17 H2 K1
      FROM    K2 K0 K2M125 K2
      MOV     K4M125 D110  ; HAMMER  MILL    AMPS
1883  LD      M8000
      RD3A    K2 K21 D110
; K1986 = 1800PSI REPLACED PUMP CHANGE OVER HMI BUTTON  D1025
1891  LD      M451  ; HAYLAGE AUTO    PAGE
      OR      M513  ; HAYLAGE RUNNING
      OR      M466  ; HAYLAGE SETTINGSPAGE
      MPS
      AND>    D100 K1986  ; PRESURE
      OUT     M470  ; PRESURE SWITCH  ROUND
      MRD
      AND>    D101 D1005  ; WEIGHT / HMI SET POINT 1
      OUT     M150  ; HAYLAGE SET     POINT 1
      MRD
      AND>    D101 D1010  ; WEIGHT / HMI SET POINT 2
      OUT     M151  ; HAYLAGE SET     POINT 2
      MRD
      AND>    D101 D1015  ; WEIGHT / HMI SET POINT 3
      OUT     M152  ; HAYLAGE SET     POINT 3
      MRD
      AND>    D101 D1110  ; WEIGHT / HMI SET POINT 4 HAYLAGE
      OUT     M545  ; HAYLAGE SET     POINT 4
      MRD
      AND>    D101 D1020  ; WEIGHT / HMI     O/WIEGHTHAYLAGE
      OUT     M153  ; HAYLAGE O/WIEGHTSET     POINT
      MRD
      AND>    D101 D1050  ; WEIGHT / WEIGHT  STILL   ON      CONVEYOR
      OUT     M154  ; WEIGHT  STILL ONCONVEYORHAYLAGE
      MPP
      AND>    D101 D3035  ; WEIGHT / WEIGHT  REACHED HAYLAGE SLOWDWN
      OUT     M800  ; HAYLAGE WEIGHT  SLOW    DOWN
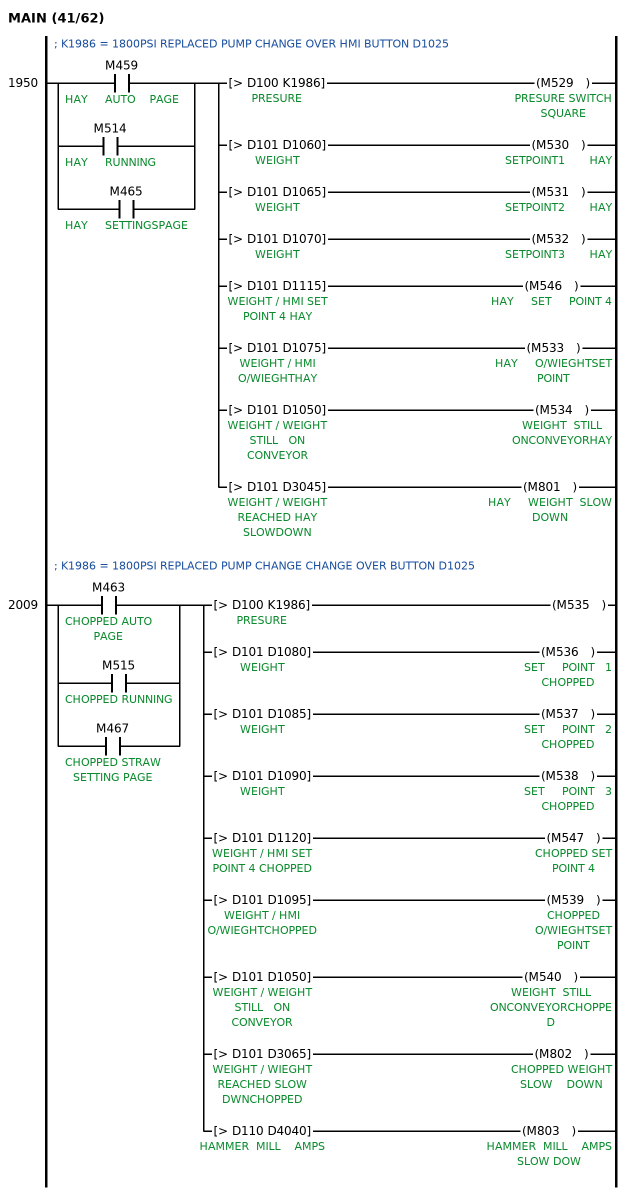
; K1986 = 1800PSI REPLACED PUMP CHANGE OVER HMI BUTTON D1025
1950  LD      M459  ; HAY     AUTO    PAGE
      OR      M514  ; HAY     RUNNING
      OR      M465  ; HAY     SETTINGSPAGE
      MPS
      AND>    D100 K1986  ; PRESURE
      OUT     M529  ; PRESURE SWITCH  SQUARE
      MRD
      AND>    D101 D1060  ; WEIGHT
      OUT     M530  ; SETPOINT1       HAY
      MRD
      AND>    D101 D1065  ; WEIGHT
      OUT     M531  ; SETPOINT2       HAY
      MRD
      AND>    D101 D1070  ; WEIGHT
      OUT     M532  ; SETPOINT3       HAY
      MRD
      AND>    D101 D1115  ; WEIGHT / HMI SET POINT 4 HAY
      OUT     M546  ; HAY     SET     POINT 4
      MRD
      AND>    D101 D1075  ; WEIGHT / HMI     O/WIEGHTHAY
      OUT     M533  ; HAY     O/WIEGHTSET     POINT
      MRD
      AND>    D101 D1050  ; WEIGHT / WEIGHT  STILL   ON      CONVEYOR
      OUT     M534  ; WEIGHT  STILL ONCONVEYORHAY
      MPP
      AND>    D101 D3045  ; WEIGHT / WEIGHT  REACHED HAY SLOWDOWN
      OUT     M801  ; HAY     WEIGHT  SLOW    DOWN
; K1986 = 1800PSI REPLACED PUMP CHANGE CHANGE OVER BUTTON D1025
2009  LD      M463  ; CHOPPED AUTO    PAGE
      OR      M515  ; CHOPPED RUNNING
      OR      M467  ; CHOPPED STRAW   SETTING PAGE
      MPS
      AND>    D100 K1986  ; PRESURE
      OUT     M535
      MRD
      AND>    D101 D1080  ; WEIGHT
      OUT     M536  ; SET     POINT   1       CHOPPED
      MRD
      AND>    D101 D1085  ; WEIGHT
      OUT     M537  ; SET     POINT   2       CHOPPED
      MRD
      AND>    D101 D1090  ; WEIGHT
      OUT     M538  ; SET     POINT   3       CHOPPED
      MRD
      AND>    D101 D1120  ; WEIGHT / HMI SET POINT 4 CHOPPED
      OUT     M547  ; CHOPPED SET     POINT 4
      MRD
      AND>    D101 D1095  ; WEIGHT / HMI     O/WIEGHTCHOPPED
      OUT     M539  ; CHOPPED O/WIEGHTSET     POINT
      MRD
      AND>    D101 D1050  ; WEIGHT / WEIGHT  STILL   ON      CONVEYOR
      OUT     M540  ; WEIGHT  STILL ONCONVEYORCHOPPED
      MRD
      AND>    D101 D3065  ; WEIGHT / WIEGHT  REACHED SLOW DWNCHOPPED
      OUT     M802  ; CHOPPED WEIGHT  SLOW    DOWN
      MPP
      AND>    D110 D4040  ; HAMMER  MILL    AMPS
      OUT     M803  ; HAMMER  MILL    AMPS    SLOW DOW
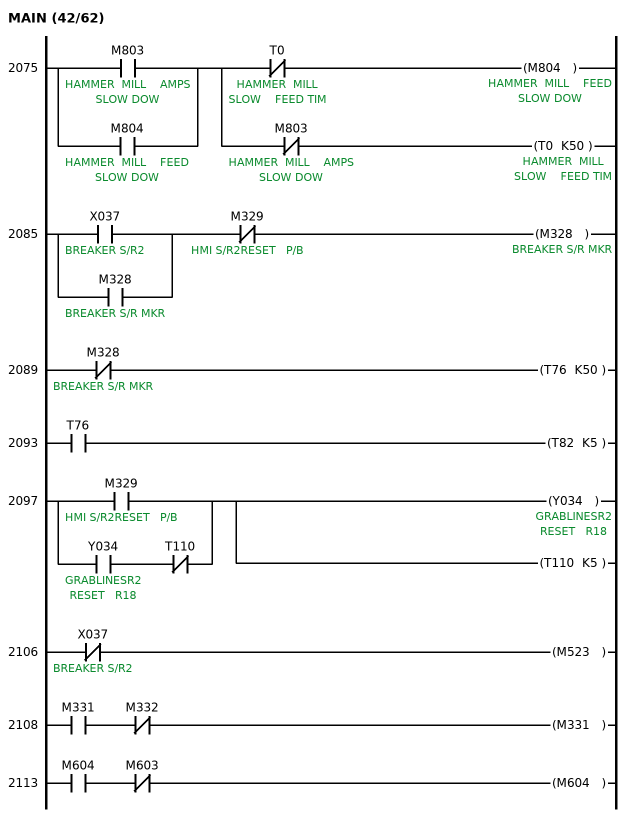
2075  LD      M803  ; HAMMER  MILL    AMPS    SLOW DOW
      OR      M804  ; HAMMER  MILL    FEED    SLOW DOW
      MPS
      ANI     T0  ; HAMMER  MILL    SLOW    FEED TIM
      OUT     M804  ; HAMMER  MILL    FEED    SLOW DOW
      MPP
      ANI     M803  ; HAMMER  MILL    AMPS    SLOW DOW
      OUT     T0 K50  ; HAMMER  MILL    SLOW    FEED TIM
2085  LD      X037  ; BREAKER S/R2
      OR      M328  ; BREAKER S/R MKR
      ANI     M329  ; HMI S/R2RESET   P/B
      OUT     M328  ; BREAKER S/R MKR
2089  LDI     M328  ; BREAKER S/R MKR
      OUT     T76 K50
2093  LD      T76
      OUT     T82 K5
2097  LD      M329  ; HMI S/R2RESET   P/B
      LD      Y034  ; GRABLINESR2     RESET   R18
      ANI     T110
      ORB
      OUT     Y034  ; GRABLINESR2     RESET   R18
      OUT     T110 K5
2106  LDI     X037  ; BREAKER S/R2
      OUT     M523
2108  LD      M331
      ANI     M332
      OUT     M331
2113  LD      M604
      ANI     M603
      OUT     M604
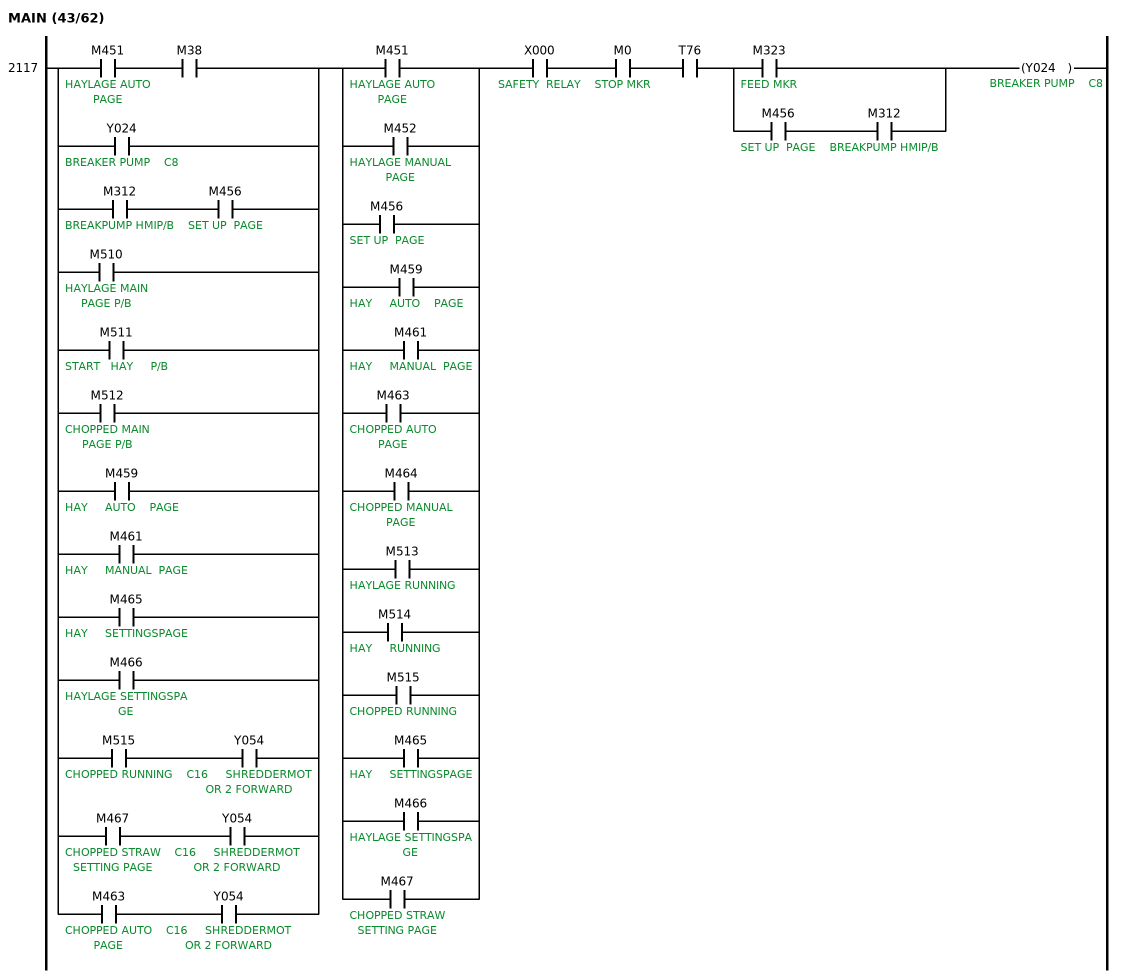
2117  LD      M451  ; HAYLAGE AUTO    PAGE
      AND     M38
      OR      Y024  ; BREAKER PUMP    C8
      LD      M312  ; BREAKPUMP HMIP/B
      AND     M456  ; SET UP  PAGE
      ORB
      OR      M510  ; HAYLAGE MAIN    PAGE P/B
      OR      M511  ; START   HAY     P/B
      OR      M512  ; CHOPPED MAIN    PAGE P/B
      OR      M459  ; HAY     AUTO    PAGE
      OR      M461  ; HAY     MANUAL  PAGE
      OR      M465  ; HAY     SETTINGSPAGE
      OR      M466  ; HAYLAGE SETTINGSPAGE
      LD      M515  ; CHOPPED RUNNING
      AND     Y054  ; C16     SHREDDERMOTOR 2 FORWARD
      ORB
      LD      M467  ; CHOPPED STRAW   SETTING PAGE
      AND     Y054  ; C16     SHREDDERMOTOR 2 FORWARD
      ORB
      LD      M463  ; CHOPPED AUTO    PAGE
      AND     Y054  ; C16     SHREDDERMOTOR 2 FORWARD
      ORB
      LD      M451  ; HAYLAGE AUTO    PAGE
      OR      M452  ; HAYLAGE MANUAL  PAGE
      OR      M456  ; SET UP  PAGE
      OR      M459  ; HAY     AUTO    PAGE
      OR      M461  ; HAY     MANUAL  PAGE
      OR      M463  ; CHOPPED AUTO    PAGE
      OR      M464  ; CHOPPED MANUAL  PAGE
      OR      M513  ; HAYLAGE RUNNING
      OR      M514  ; HAY     RUNNING
      OR      M515  ; CHOPPED RUNNING
      OR      M465  ; HAY     SETTINGSPAGE
      OR      M466  ; HAYLAGE SETTINGSPAGE
      OR      M467  ; CHOPPED STRAW   SETTING PAGE
      ANB
      AND     X000  ; SAFETY  RELAY
      AND     M0  ; STOP MKR
      AND     T76
      LD      M323  ; FEED MKR
      LD      M456  ; SET UP  PAGE
      AND     M312  ; BREAKPUMP HMIP/B
      ORB
      ANB
      OUT     Y024  ; BREAKER PUMP    C8
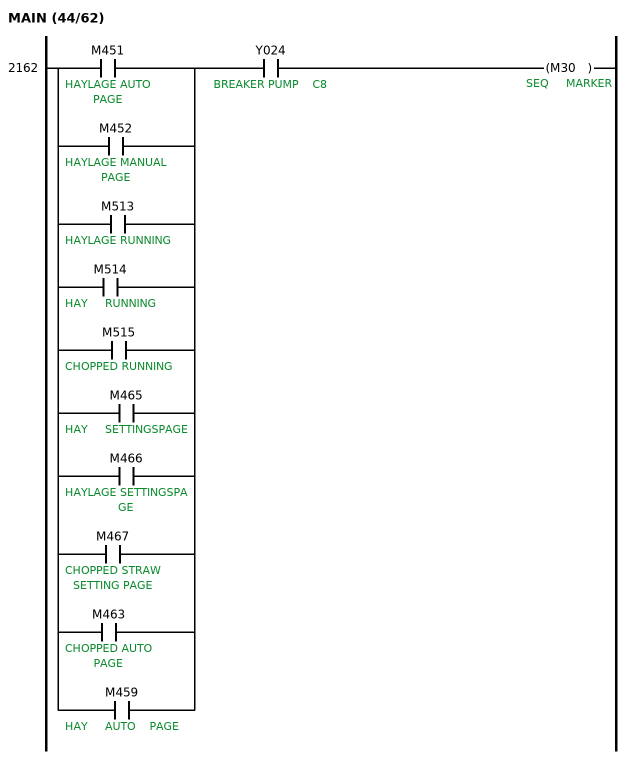
2162  LD      M451  ; HAYLAGE AUTO    PAGE
      OR      M452  ; HAYLAGE MANUAL  PAGE
      OR      M513  ; HAYLAGE RUNNING
      OR      M514  ; HAY     RUNNING
      OR      M515  ; CHOPPED RUNNING
      OR      M465  ; HAY     SETTINGSPAGE
      OR      M466  ; HAYLAGE SETTINGSPAGE
      OR      M467  ; CHOPPED STRAW   SETTING PAGE
      OR      M463  ; CHOPPED AUTO    PAGE
      OR      M459  ; HAY     AUTO    PAGE
      AND     Y024  ; BREAKER PUMP    C8
      OUT     M30  ; SEQ     MARKER
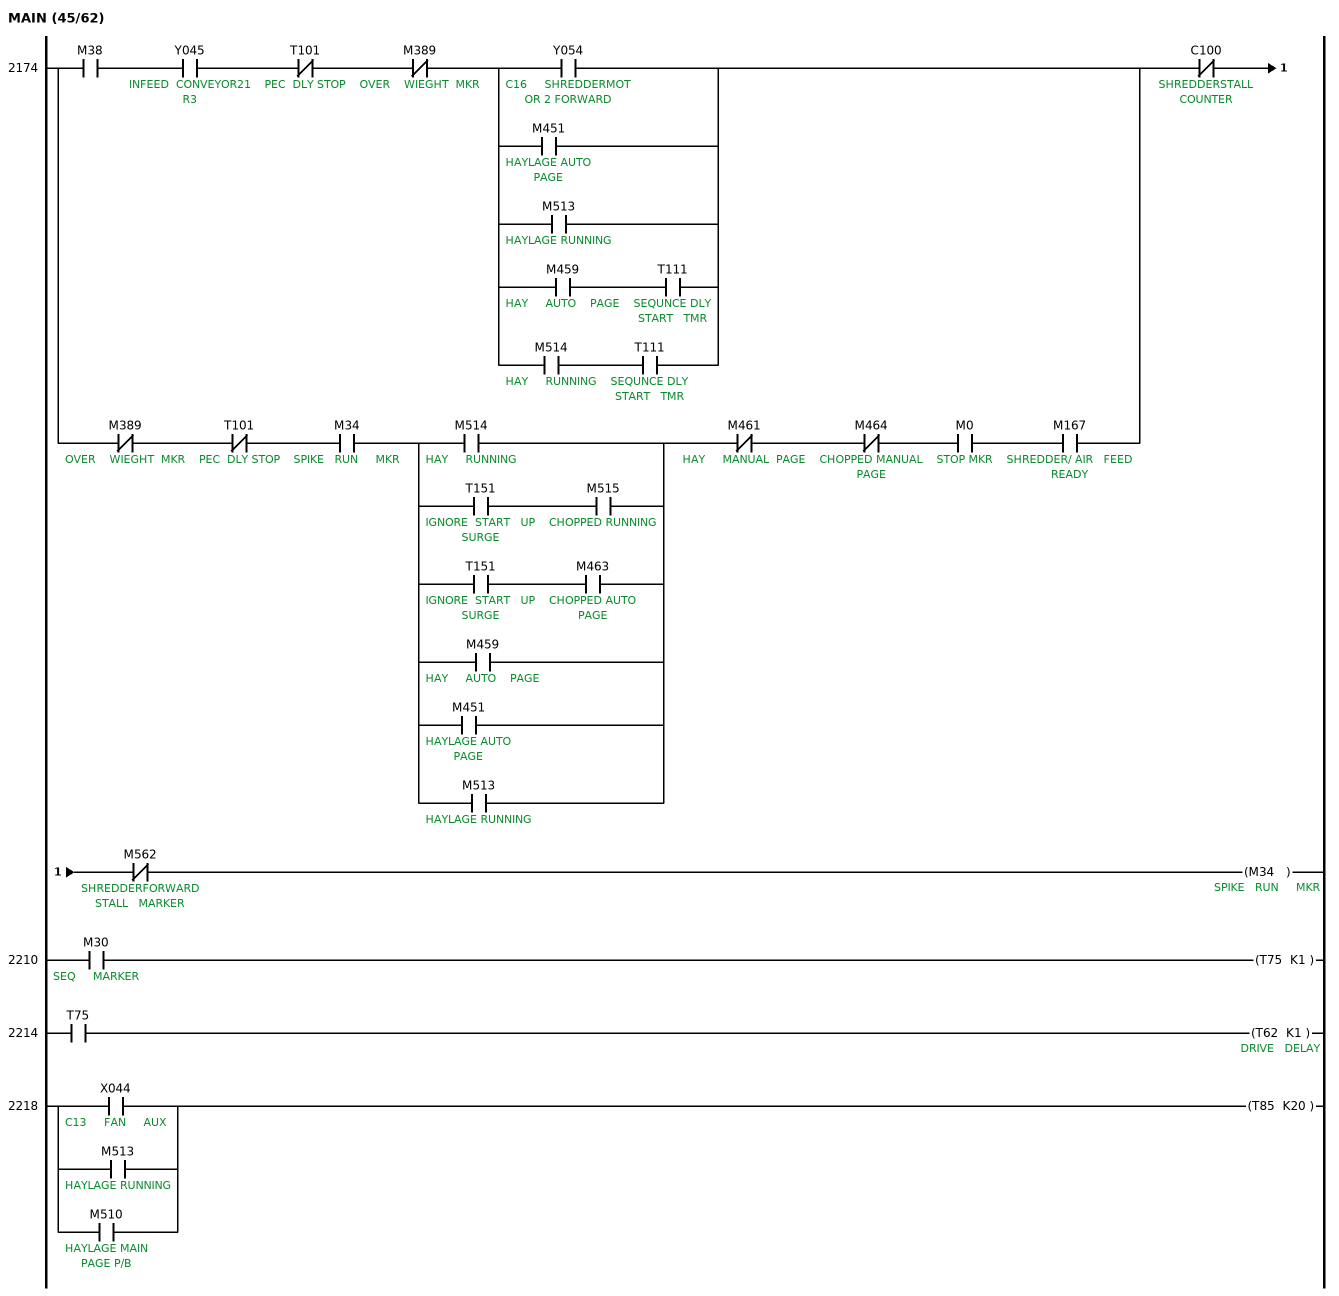
2174  LD      M38
      AND     Y045  ; INFEED  CONVEYOR21R3
      ANI     T101  ; PEC  DLY STOP
      ANI     M389  ; OVER    WIEGHT  MKR
      LD      Y054  ; C16     SHREDDERMOTOR 2 FORWARD
      OR      M451  ; HAYLAGE AUTO    PAGE
      OR      M513  ; HAYLAGE RUNNING
      LD      M459  ; HAY     AUTO    PAGE
      AND     T111  ; SEQUNCE DLY     START   TMR
      ORB
      LD      M514  ; HAY     RUNNING
      AND     T111  ; SEQUNCE DLY     START   TMR
      ORB
      ANB
      LDI     M389  ; OVER    WIEGHT  MKR
      ANI     T101  ; PEC  DLY STOP
      AND     M34  ; SPIKE   RUN     MKR
      LD      M514  ; HAY     RUNNING
      LD      T151  ; IGNORE  START   UP      SURGE
      AND     M515  ; CHOPPED RUNNING
      ORB
      LD      T151  ; IGNORE  START   UP      SURGE
      AND     M463  ; CHOPPED AUTO    PAGE
      ORB
      OR      M459  ; HAY     AUTO    PAGE
      OR      M451  ; HAYLAGE AUTO    PAGE
      OR      M513  ; HAYLAGE RUNNING
      ANB
      ANI     M461  ; HAY     MANUAL  PAGE
      ANI     M464  ; CHOPPED MANUAL  PAGE
      AND     M0  ; STOP MKR
      AND     M167  ; SHREDDER/ AIR   FEED    READY
      ORB
      ANI     C100  ; SHREDDERSTALL   COUNTER
      ANI     M562  ; SHREDDERFORWARD STALL   MARKER
      OUT     M34  ; SPIKE   RUN     MKR
2210  LD      M30  ; SEQ     MARKER
      OUT     T75 K1
2214  LD      T75
      OUT     T62 K1  ; DRIVE   DELAY
2218  LD      X044  ; C13     FAN     AUX
      OR      M513  ; HAYLAGE RUNNING
      OR      M510  ; HAYLAGE MAIN    PAGE P/B
      OUT     T85 K20
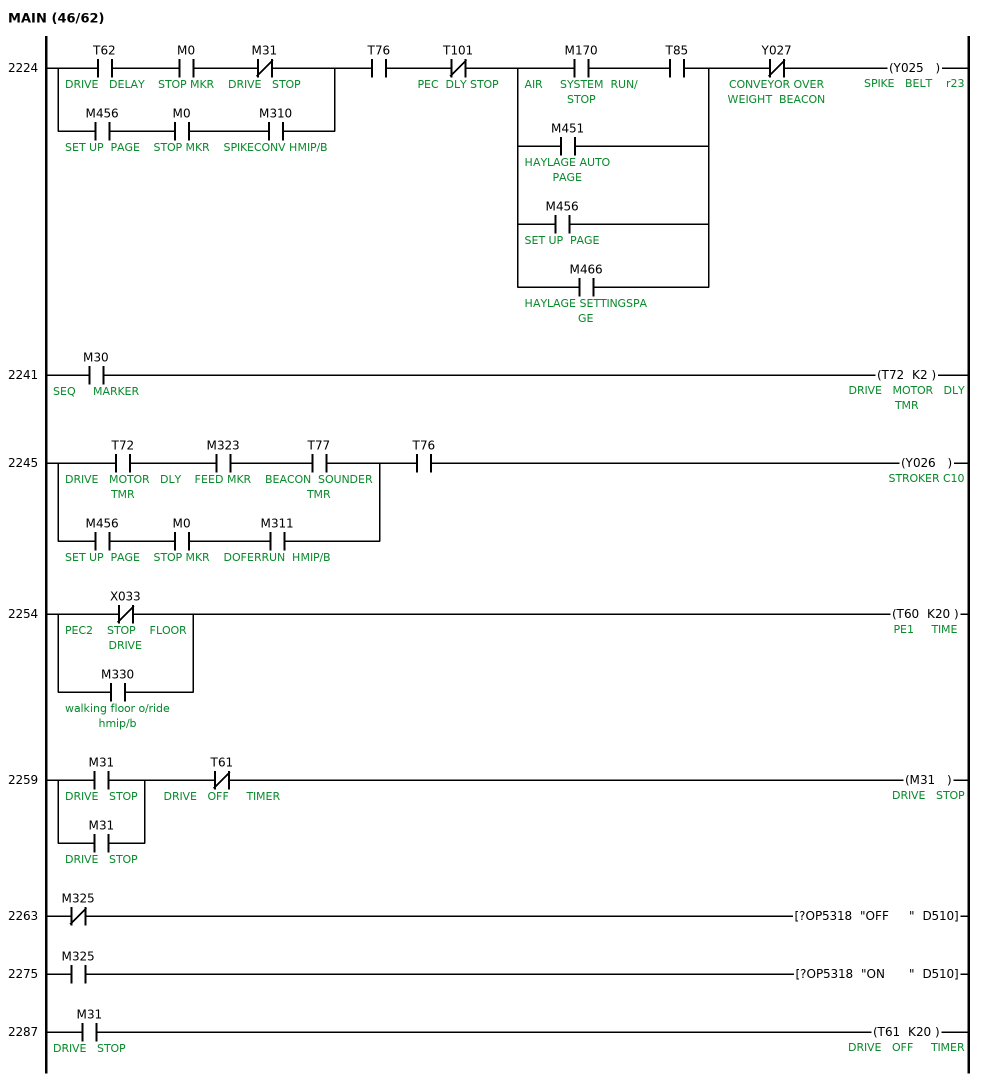
2224  LD      T62  ; DRIVE   DELAY
      AND     M0  ; STOP MKR
      ANI     M31  ; DRIVE   STOP
      LD      M456  ; SET UP  PAGE
      AND     M0  ; STOP MKR
      AND     M310  ; SPIKECONV HMIP/B
      ORB
      AND     T76
      ANI     T101  ; PEC  DLY STOP
      LD      M170  ; AIR     SYSTEM  RUN/    STOP
      AND     T85
      OR      M451  ; HAYLAGE AUTO    PAGE
      OR      M456  ; SET UP  PAGE
      OR      M466  ; HAYLAGE SETTINGSPAGE
      ANB
      ANI     Y027  ; CONVEYOR OVER   WEIGHT  BEACON
      OUT     Y025  ; SPIKE   BELT    r23
2241  LD      M30  ; SEQ     MARKER
      OUT     T72 K2  ; DRIVE   MOTOR   DLY TMR
2245  LD      T72  ; DRIVE   MOTOR   DLY TMR
      AND     M323  ; FEED MKR
      AND     T77  ; BEACON  SOUNDER TMR
      LD      M456  ; SET UP  PAGE
      AND     M0  ; STOP MKR
      AND     M311  ; DOFERRUN  HMIP/B
      ORB
      AND     T76
      OUT     Y026  ; STROKER C10
2254  LDI     X033  ; PEC2    STOP    FLOOR   DRIVE
      OR      M330  ; walking floor o/ride hmip/b
      OUT     T60 K20  ; PE1     TIME
2259  LD      M31  ; DRIVE   STOP
      OR      M31  ; DRIVE   STOP
      ANI     T61  ; DRIVE   OFF     TIMER
      OUT     M31  ; DRIVE   STOP
2263  LDI     M325
      ?OP5318 "OFF     " D510
2275  LD      M325
      ?OP5318 "ON      " D510
2287  LD      M31  ; DRIVE   STOP
      OUT     T61 K20  ; DRIVE   OFF     TIMER
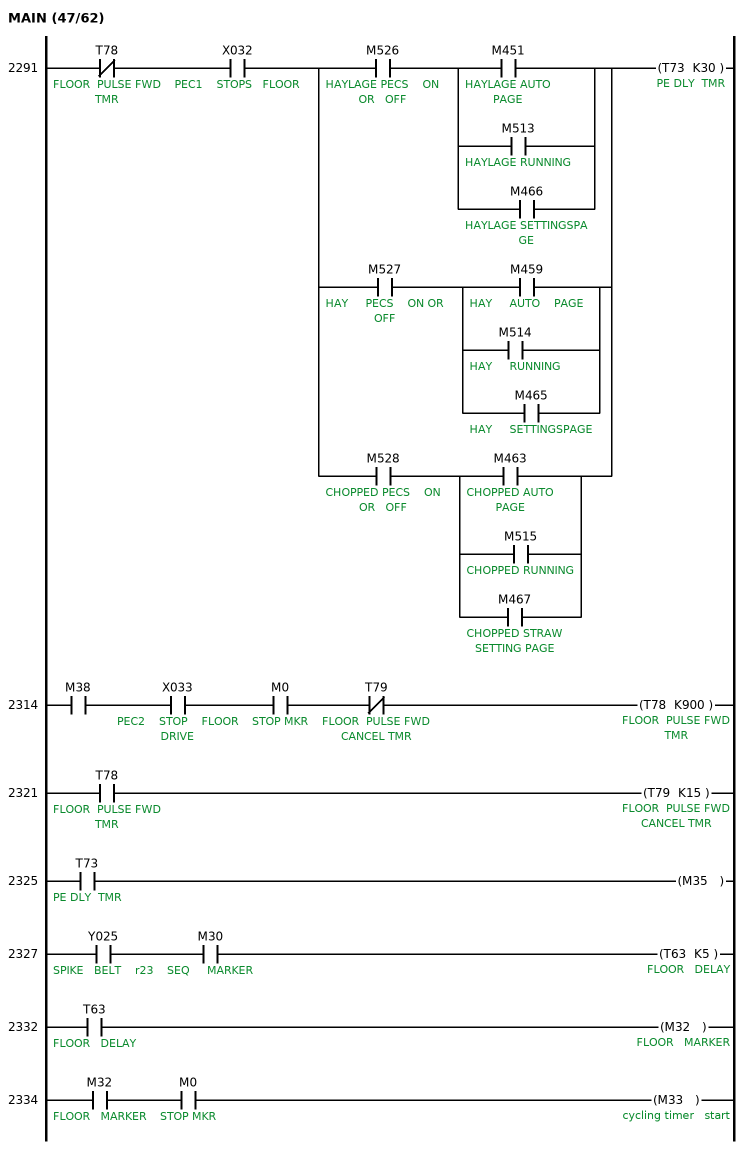
2291  LDI     T78  ; FLOOR  PULSE FWD TMR
      AND     X032  ; PEC1    STOPS   FLOOR
      LD      M526  ; HAYLAGE PECS    ON OR   OFF
      LD      M451  ; HAYLAGE AUTO    PAGE
      OR      M513  ; HAYLAGE RUNNING
      OR      M466  ; HAYLAGE SETTINGSPAGE
      ANB
      LD      M527  ; HAY     PECS    ON OR   OFF
      LD      M459  ; HAY     AUTO    PAGE
      OR      M514  ; HAY     RUNNING
      OR      M465  ; HAY     SETTINGSPAGE
      ANB
      ORB
      LD      M528  ; CHOPPED PECS    ON OR   OFF
      LD      M463  ; CHOPPED AUTO    PAGE
      OR      M515  ; CHOPPED RUNNING
      OR      M467  ; CHOPPED STRAW   SETTING PAGE
      ANB
      ORB
      ANB
      OUT     T73 K30  ; PE DLY  TMR
2314  LD      M38
      AND     X033  ; PEC2    STOP    FLOOR   DRIVE
      AND     M0  ; STOP MKR
      ANI     T79  ; FLOOR  PULSE FWD CANCEL TMR
      OUT     T78 K900  ; FLOOR  PULSE FWD TMR
2321  LD      T78  ; FLOOR  PULSE FWD TMR
      OUT     T79 K15  ; FLOOR  PULSE FWD CANCEL TMR
2325  LD      T73  ; PE DLY  TMR
      OUT     M35
2327  LD      Y025  ; SPIKE   BELT    r23
      AND     M30  ; SEQ     MARKER
      OUT     T63 K5  ; FLOOR   DELAY
2332  LD      T63  ; FLOOR   DELAY
      OUT     M32  ; FLOOR   MARKER
2334  LD      M32  ; FLOOR   MARKER
      AND     M0  ; STOP MKR
      OUT     M33  ; cycling timer   start
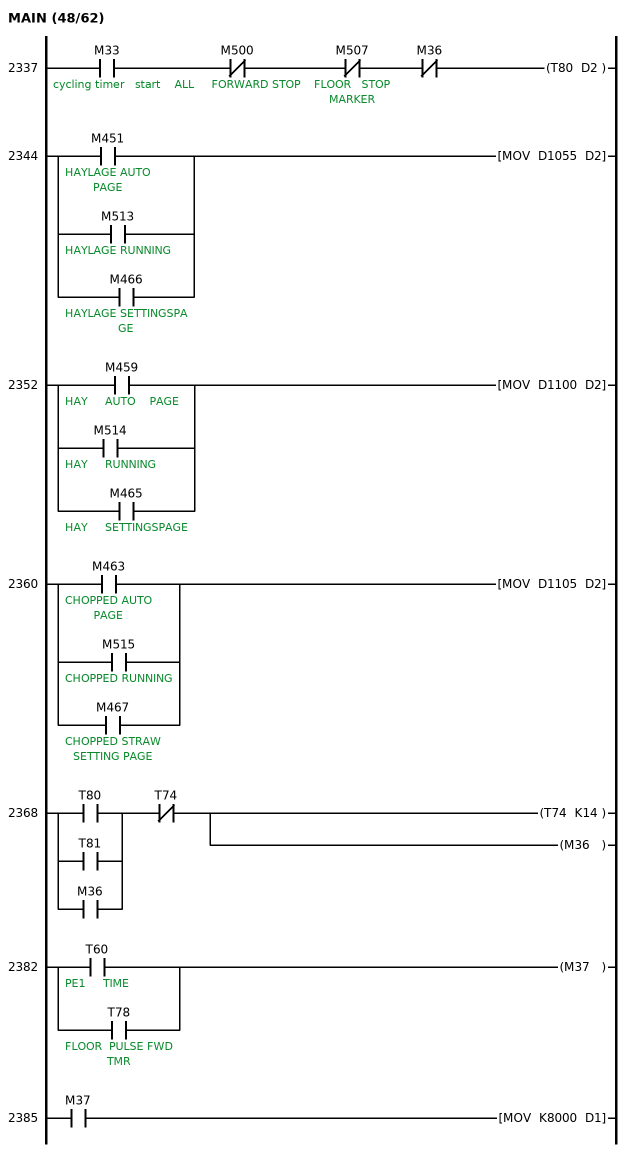
2337  LD      M33  ; cycling timer   start
      ANI     M500  ; ALL     FORWARD STOP
      ANI     M507  ; FLOOR   STOP    MARKER
      ANI     M36
      OUT     T80 D2
2344  LD      M451  ; HAYLAGE AUTO    PAGE
      OR      M513  ; HAYLAGE RUNNING
      OR      M466  ; HAYLAGE SETTINGSPAGE
      MOV     D1055 D2
2352  LD      M459  ; HAY     AUTO    PAGE
      OR      M514  ; HAY     RUNNING
      OR      M465  ; HAY     SETTINGSPAGE
      MOV     D1100 D2
2360  LD      M463  ; CHOPPED AUTO    PAGE
      OR      M515  ; CHOPPED RUNNING
      OR      M467  ; CHOPPED STRAW   SETTING PAGE
      MOV     D1105 D2
2368  LD      T80
      OR      T81
      OR      M36
      ANI     T74
      OUT     T74 K14
      OUT     M36
2382  LD      T60  ; PE1     TIME
      OR      T78  ; FLOOR  PULSE FWD TMR
      OUT     M37
2385  LD      M37
      MOV     K8000 D1
